LIN {X 0,Y 453.671,Z 73.472,A -85,B 0,C 180,E1 -8454.666,E2 -8454.666} C_VEL
LIN {X 0,Y 453.744,Z 73.459,A -85,B 0,C 180,E1 -8457.336,E2 -8457.336} C_VEL
LIN {X 0,Y 453.822,Z 73.438,A -85,B 0,C 180,E1 -8460,E2 -8460} C_VEL
LIN {X 0,Y 453.744,Z 73.457,A -85,B 0,C 180,E1 -8462.663,E2 -8462.663} C_VEL
LIN {X 0,Y 453.677,Z 73.469,A -85,B 0,C 180,E1 -8466.225,E2 -8466.225} C_VEL
LIN {X 0,Y 453.591,Z 73.469,A -85,B 0,C 180,E1 -8468.913,E2 -8468.913} C_VEL
LIN {X 0,Y 453.601,Z 73.475,A -85,B 0,C 180,E1 -8472.55,E2 -8472.55} C_VEL
LIN {X 0,Y 453.543,Z 73.483,A -85,B 0,C 180,E1 -8476.195,E2 -8476.195} C_VEL
LIN {X 0,Y 453.518,Z 73.478,A -85,B 0,C 180,E1 -8479.04,E2 -8479.04} C_VEL
LIN {X 0,Y 453.475,Z 73.495,A -85,B 0,C 180,E1 -8481.836,E2 -8481.836} C_VEL
LIN {X 0,Y 453.512,Z 73.492,A -85,B 0,C 180,E1 -8484.734,E2 -8484.734} C_VEL
LIN {X 0,Y 453.535,Z 73.478,A -85,B 0,C 180,E1 -8487.96,E2 -8487.96} C_VEL
LIN {X 0,Y 453.464,Z 73.497,A -85,B 0,C 180,E1 -8491.525,E2 -8491.525} C_VEL
LIN {X 0,Y 453.486,Z 73.489,A -85,B 0,C 180,E1 -8494.777,E2 -8494.777} C_VEL
LIN {X 0,Y 453.477,Z 73.498,A -85,B 0,C 180,E1 -8498.31,E2 -8498.31} C_VEL
LIN {X 0,Y 453.513,Z 73.488,A -85,B 0,C 180,E1 -8500.606,E2 -8500.606} C_VEL
LIN {X 0,Y 453.463,Z 73.501,A -85,B 0,C 180,E1 -8504.221,E2 -8504.221} C_VEL
LIN {X 0,Y 453.458,Z 73.476,A -85,B 0,C 180,E1 -8507.005,E2 -8507.005} C_VEL
LIN {X 0,Y 453.502,Z 73.493,A -85,B 0,C 180,E1 -8510.552,E2 -8510.552} C_VEL
LIN {X 0,Y 453.454,Z 73.495,A -85,B 0,C 180,E1 -8513.917,E2 -8513.917} C_VEL
LIN {X 0,Y 453.479,Z 73.493,A -85,B 0,C 180,E1 -8517.151,E2 -8517.151} C_VEL
LIN {X 0,Y 453.471,Z 73.488,A -85,B 0,C 180,E1 -8520.268,E2 -8520.268} C_VEL
LIN {X 0,Y 453.506,Z 73.494,A -85,B 0,C 180,E1 -8523.294,E2 -8523.294} C_VEL
LIN {X 0,Y 453.5,Z 73.496,A -85,B 0,C 180,E1 -8526.239,E2 -8526.239} C_VEL
LIN {X 0,Y 453.48,Z 73.498,A -85,B 0,C 180,E1 -8529.118,E2 -8529.118} C_VEL
LIN {X 0,Y 453.509,Z 73.497,A -85,B 0,C 180,E1 -8531.945,E2 -8531.945} C_VEL
LIN {X 0,Y 453.538,Z 73.491,A -85,B 0,C 180,E1 -8534.726,E2 -8534.726} C_VEL
LIN {X 0,Y 453.557,Z 73.488,A -85,B 0,C 180,E1 -8538.379,E2 -8538.379} C_VEL
LIN {X 0,Y 453.649,Z 73.478,A -85,B 0,C 180,E1 -8541.985,E2 -8541.985} C_VEL
LIN {X 0,Y 453.634,Z 73.479,A -85,B 0,C 180,E1 -8543.083,E2 -8543.083} C_VEL
LIN {X 0,Y 452.949,Z 73.565,A -85,B 0,C 180,E1 -8543.824,E2 -8543.824} C_VEL
LIN {X 0,Y 449.999,Z 73.934,A -85,B 0,C 180,E1 -8545.025,E2 -8545.025} C_VEL
LIN {X 0,Y 447.575,Z 74.234,A -85,B 0,C 180,E1 -8545.995,E2 -8545.995} C_VEL
LIN {X 0,Y 446.638,Z 74.352,A -85,B 0,C 180,E1 -8546.745,E2 -8546.745} C_VEL
LIN {X 0,Y 446.618,Z 74.353,A -85,B 0,C 180,E1 -8546.999,E2 -8546.999} C_VEL
LIN {X 0,Y 446.791,Z 74.332,A -85,B 0,C 180,E1 -8550,E2 -8550} C_VEL
LIN {X 0,Y 446.706,Z 74.344,A -85,B 0,C 180,E1 -8552.705,E2 -8552.705} C_VEL
LIN {X 0,Y 446.645,Z 74.351,A -85,B 0,C 180,E1 -8556.324,E2 -8556.324} C_VEL
LIN {X 0,Y 446.535,Z 74.365,A -85,B 0,C 180,E1 -8559.055,E2 -8559.055} C_VEL
LIN {X 0,Y 446.518,Z 74.367,A -85,B 0,C 180,E1 -8562.73,E2 -8562.73} C_VEL
LIN {X 0,Y 446.493,Z 74.371,A -85,B 0,C 180,E1 -8566.228,E2 -8566.228} C_VEL
LIN {X 0,Y 446.466,Z 74.371,A -85,B 0,C 180,E1 -8569.303,E2 -8569.303} C_VEL
LIN {X 0,Y 446.416,Z 74.381,A -85,B 0,C 180,E1 -8572.2,E2 -8572.2} C_VEL
LIN {X 0,Y 446.454,Z 74.371,A -85,B 0,C 180,E1 -8575.152,E2 -8575.152} C_VEL
LIN {X 0,Y 446.481,Z 74.364,A -85,B 0,C 180,E1 -8578.179,E2 -8578.179} C_VEL
LIN {X 0,Y 446.431,Z 74.378,A -85,B 0,C 180,E1 -8581.778,E2 -8581.778} C_VEL
LIN {X 0,Y 446.427,Z 74.353,A -85,B 0,C 180,E1 -8585.054,E2 -8585.054} C_VEL
LIN {X 0,Y 446.427,Z 74.377,A -85,B 0,C 180,E1 -8588.082,E2 -8588.082} C_VEL
LIN {X 0,Y 446.423,Z 74.361,A -85,B 0,C 180,E1 -8590.918,E2 -8590.918} C_VEL
LIN {X 0,Y 446.396,Z 74.367,A -85,B 0,C 180,E1 -8593.846,E2 -8593.846} C_VEL
LIN {X 0,Y 446.396,Z 74.377,A -85,B 0,C 180,E1 -8596.404,E2 -8596.404} C_VEL
LIN {X 0,Y 446.464,Z 74.367,A -85,B 0,C 180,E1 -8599.805,E2 -8599.805} C_VEL
LIN {X 0,Y 446.428,Z 74.374,A -85,B 0,C 180,E1 -8602.124,E2 -8602.124} C_VEL
LIN {X 0,Y 446.428,Z 74.367,A -85,B 0,C 180,E1 -8605.478,E2 -8605.478} C_VEL
LIN {X 0,Y 446.414,Z 74.377,A -85,B 0,C 180,E1 -8608.7,E2 -8608.7} C_VEL
LIN {X 0,Y 446.482,Z 74.357,A -85,B 0,C 180,E1 -8611.822,E2 -8611.822} C_VEL
LIN {X 0,Y 446.456,Z 74.369,A -85,B 0,C 180,E1 -8614.848,E2 -8614.848} C_VEL
LIN {X 0,Y 446.446,Z 74.371,A -85,B 0,C 180,E1 -8618.245,E2 -8618.245} C_VEL
LIN {X 0,Y 446.455,Z 74.356,A -85,B 0,C 180,E1 -8621.65,E2 -8621.65} C_VEL
LIN {X 0,Y 446.506,Z 74.366,A -85,B 0,C 180,E1 -8624.48,E2 -8624.48} C_VEL
LIN {X 0,Y 446.538,Z 74.357,A -85,B 0,C 180,E1 -8628.194,E2 -8628.194} C_VEL
LIN {X 0,Y 446.599,Z 74.341,A -85,B 0,C 180,E1 -8631.858,E2 -8631.858} C_VEL
LIN {X 0,Y 446.645,Z 74.349,A -85,B 0,C 180,E1 -8634.583,E2 -8634.583} C_VEL
LIN {X 0,Y 446.664,Z 74.335,A -85,B 0,C 180,E1 -8638.197,E2 -8638.197} C_VEL
LIN {X 0,Y 446.792,Z 74.312,A -85,B 0,C 180,E1 -8640,E2 -8640} C_VEL
LIN {X 0,Y 446.691,Z 74.337,A -85,B 0,C 180,E1 -8642.706,E2 -8642.706} C_VEL
LIN {X 0,Y 446.647,Z 74.344,A -85,B 0,C 180,E1 -8646.324,E2 -8646.324} C_VEL
LIN {X 0,Y 446.538,Z 74.346,A -85,B 0,C 180,E1 -8649.056,E2 -8649.056} C_VEL
LIN {X 0,Y 446.522,Z 74.357,A -85,B 0,C 180,E1 -8652.73,E2 -8652.73} C_VEL
LIN {X 0,Y 446.497,Z 74.359,A -85,B 0,C 180,E1 -8656.228,E2 -8656.228} C_VEL
LIN {X 0,Y 446.47,Z 74.354,A -85,B 0,C 180,E1 -8659.304,E2 -8659.304} C_VEL
LIN {X 0,Y 446.419,Z 74.372,A -85,B 0,C 180,E1 -8662.2,E2 -8662.2} C_VEL
LIN {X 0,Y 446.459,Z 74.367,A -85,B 0,C 180,E1 -8665.153,E2 -8665.153} C_VEL
LIN {X 0,Y 446.486,Z 74.358,A -85,B 0,C 180,E1 -8668.179,E2 -8668.179} C_VEL
LIN {X 0,Y 446.42,Z 74.373,A -85,B 0,C 180,E1 -8671.775,E2 -8671.775} C_VEL
LIN {X 0,Y 446.43,Z 74.364,A -85,B 0,C 180,E1 -8674.523,E2 -8674.523} C_VEL
LIN {X 0,Y 446.415,Z 74.375,A -85,B 0,C 180,E1 -8678.079,E2 -8678.079} C_VEL
LIN {X 0,Y 446.428,Z 74.373,A -85,B 0,C 180,E1 -8680.918,E2 -8680.918} C_VEL
LIN {X 0,Y 446.401,Z 74.376,A -85,B 0,C 180,E1 -8683.847,E2 -8683.847} C_VEL
LIN {X 0,Y 446.4,Z 74.381,A -85,B 0,C 180,E1 -8686.404,E2 -8686.404} C_VEL
LIN {X 0,Y 446.428,Z 74.361,A -85,B 0,C 180,E1 -8689.083,E2 -8689.083} C_VEL
LIN {X 0,Y 446.429,Z 74.376,A -85,B 0,C 180,E1 -8692.123,E2 -8692.123} C_VEL
LIN {X 0,Y 446.432,Z 74.37,A -85,B 0,C 180,E1 -8695.477,E2 -8695.477} C_VEL
LIN {X 0,Y 446.419,Z 74.377,A -85,B 0,C 180,E1 -8698.7,E2 -8698.7} C_VEL
LIN {X 0,Y 446.548,Z 74.569,A -85,B 0,C 180,E1 -8701.867,E2 -8701.867} C_VEL
LIN {X 0,Y 448.347,Z 84.511,A -85,B 0,C 180,E1 -8704.464,E2 -8704.464} C_VEL
LIN {X 0,Y 448.456,Z 88.047,A -85,B 0,C 180,E1 -8705.362,E2 -8705.362} C_VEL
LIN {X 0,Y 447.632,Z 102.965,A -85,B 0,C 180,E1 -8708.832,E2 -8708.832} C_VEL
LIN {X 0,Y 447.004,Z 115.084,A -85,B 0,C 180,E1 -8711.673,E2 -8711.673} C_VEL
LIN {X 0,Y 446.957,Z 117.073,A -85,B 0,C 180,E1 -8712.115,E2 -8712.115} C_VEL
LIN {X 0,Y 447.469,Z 120.446,A -85,B 0,C 180,E1 -8712.243,E2 -8712.243} C_VEL
LIN {X 0,Y 450.806,Z 140.583,A -85,B 0,C 180,E1 -8712.706,E2 -8712.706} C_VEL
LIN {X 0,Y 450.052,Z 221.953,A -85,B 0,C 180,E1 -8714.024,E2 -8714.024} C_VEL
LIN {X 0,Y 449.783,Z 231.85,A -85,B 0,C 180,E1 -8714.276,E2 -8714.276} C_VEL
LIN {X 0,Y 449.405,Z 241.826,A -85,B 0,C 180,E1 -8714.64,E2 -8714.64} C_VEL
LIN {X 0,Y 448.986,Z 252.191,A -85,B 0,C 180,E1 -8715.148,E2 -8715.148} C_VEL
LIN {X 0,Y 448.514,Z 261.326,A -85,B 0,C 180,E1 -8715.712,E2 -8715.712} C_VEL
LIN {X 0,Y 448.006,Z 270.323,A -85,B 0,C 180,E1 -8716.39,E2 -8716.39} C_VEL
LIN {X 0,Y 447.59,Z 278.193,A -85,B 0,C 180,E1 -8717.098,E2 -8717.098} C_VEL
LIN {X 0,Y 447.145,Z 286.451,A -85,B 0,C 180,E1 -8717.98,E2 -8717.98} C_VEL
LIN {X 0,Y 446.687,Z 293.671,A -85,B 0,C 180,E1 -8718.888,E2 -8718.888} C_VEL
LIN {X 0,Y 446.344,Z 299.873,A -85,B 0,C 180,E1 -8719.797,E2 -8719.797} C_VEL
LIN {X 0,Y 445.989,Z 306.41,A -85,B 0,C 180,E1 -8720.933,E2 -8720.933} C_VEL
LIN {X 0,Y 445.785,Z 310.912,A -85,B 0,C 180,E1 -8721.843,E2 -8721.843} C_VEL
LIN {X 0,Y 445.554,Z 316.557,A -85,B 0,C 180,E1 -8723.251,E2 -8723.251} C_VEL
LIN {X 0,Y 445.473,Z 320.725,A -85,B 0,C 180,E1 -8724.568,E2 -8724.568} C_VEL
LIN {X 0,Y 445.412,Z 323.089,A -85,B 0,C 180,E1 -8725.475,E2 -8725.475} C_VEL
LIN {X 0,Y 445.433,Z 326.273,A -85,B 0,C 180,E1 -8727.287,E2 -8727.287} C_VEL
LIN {X 0,Y 445.356,Z 327.327,A -85,B 0,C 180,E1 -8728.191,E2 -8728.191} C_VEL
LIN {X 0,Y 445.341,Z 327.914,A -85,B 0,C 180,E1 -8729.096,E2 -8729.096} C_VEL
LIN {X 0,Y 445.341,Z 327.914,A -85,B 0,C 180,E1 -8730.904,E2 -8730.904} C_VEL
LIN {X 0,Y 445.356,Z 327.327,A -85,B 0,C 180,E1 -8731.809,E2 -8731.809} C_VEL
LIN {X 0,Y 445.433,Z 326.273,A -85,B 0,C 180,E1 -8732.713,E2 -8732.713} C_VEL
LIN {X 0,Y 445.412,Z 323.089,A -85,B 0,C 180,E1 -8734.525,E2 -8734.525} C_VEL
LIN {X 0,Y 445.466,Z 318.987,A -85,B 0,C 180,E1 -8736.038,E2 -8736.038} C_VEL
LIN {X 0,Y 445.601,Z 314.742,A -85,B 0,C 180,E1 -8737.249,E2 -8737.249} C_VEL
LIN {X 0,Y 445.887,Z 308.722,A -85,B 0,C 180,E1 -8738.612,E2 -8738.612} C_VEL
LIN {X 0,Y 446.179,Z 302.625,A -85,B 0,C 180,E1 -8739.749,E2 -8739.749} C_VEL
LIN {X 0,Y 446.489,Z 296.924,A -85,B 0,C 180,E1 -8740.658,E2 -8740.658} C_VEL
LIN {X 0,Y 447.013,Z 288.37,A -85,B 0,C 180,E1 -8741.794,E2 -8741.794} C_VEL
LIN {X 0,Y 447.481,Z 280.189,A -85,B 0,C 180,E1 -8742.702,E2 -8742.702} C_VEL
LIN {X 0,Y 447.961,Z 271.759,A -85,B 0,C 180,E1 -8743.489,E2 -8743.489} C_VEL
LIN {X 0,Y 448.412,Z 262.957,A -85,B 0,C 180,E1 -8744.175,E2 -8744.175} C_VEL
LIN {X 0,Y 448.929,Z 253.198,A -85,B 0,C 180,E1 -8744.796,E2 -8744.796} C_VEL
LIN {X 0,Y 449.332,Z 244.402,A -85,B 0,C 180,E1 -8745.246,E2 -8745.246} C_VEL
LIN {X 0,Y 449.711,Z 234.473,A -85,B 0,C 180,E1 -8745.639,E2 -8745.639} C_VEL
LIN {X 0,Y 450.046,Z 224.618,A -85,B 0,C 180,E1 -8745.918,E2 -8745.918} C_VEL
LIN {X 0,Y 450.333,Z 200.656,A -85,B 0,C 180,E1 -8746.333,E2 -8746.333} C_VEL
LIN {X 0,Y 450.666,Z 138.88,A -85,B 0,C 180,E1 -8747.327,E2 -8747.327} C_VEL
LIN {X 0,Y 446.978,Z 117.536,A -85,B 0,C 180,E1 -8747.841,E2 -8747.841} C_VEL
LIN {X 0,Y 446.948,Z 116.116,A -85,B 0,C 180,E1 -8748.073,E2 -8748.073} C_VEL
LIN {X 0,Y 447.654,Z 103.185,A -85,B 0,C 180,E1 -8751.167,E2 -8751.167} C_VEL
LIN {X 0,Y 448.399,Z 89.526,A -85,B 0,C 180,E1 -8754.347,E2 -8754.347} C_VEL
LIN {X 0,Y 448.49,Z 85.556,A -85,B 0,C 180,E1 -8755.278,E2 -8755.278} C_VEL
LIN {X 0,Y 446.71,Z 75.373,A -85,B 0,C 180,E1 -8757.908,E2 -8757.908} C_VEL
LIN {X 0,Y 446.514,Z 74.374,A -85,B 0,C 180,E1 -8758.28,E2 -8758.28} C_VEL
LIN {X 0,Y 446.422,Z 74.373,A -85,B 0,C 180,E1 -8761.775,E2 -8761.775} C_VEL
LIN {X 0,Y 446.432,Z 74.371,A -85,B 0,C 180,E1 -8764.523,E2 -8764.523} C_VEL
LIN {X 0,Y 446.431,Z 74.373,A -85,B 0,C 180,E1 -8768.081,E2 -8768.081} C_VEL
LIN {X 0,Y 446.428,Z 74.362,A -85,B 0,C 180,E1 -8770.917,E2 -8770.917} C_VEL
LIN {X 0,Y 446.402,Z 74.378,A -85,B 0,C 180,E1 -8773.846,E2 -8773.846} C_VEL
LIN {X 0,Y 446.399,Z 74.376,A -85,B 0,C 180,E1 -8776.403,E2 -8776.403} C_VEL
LIN {X 0,Y 446.428,Z 74.374,A -85,B 0,C 180,E1 -8779.082,E2 -8779.082} C_VEL
LIN {X 0,Y 446.409,Z 74.375,A -85,B 0,C 180,E1 -8782.121,E2 -8782.121} C_VEL
LIN {X 0,Y 446.43,Z 74.364,A -85,B 0,C 180,E1 -8785.477,E2 -8785.477} C_VEL
LIN {X 0,Y 446.417,Z 74.377,A -85,B 0,C 180,E1 -8788.699,E2 -8788.699} C_VEL
LIN {X 0,Y 446.486,Z 74.358,A -85,B 0,C 180,E1 -8791.821,E2 -8791.821} C_VEL
LIN {X 0,Y 446.459,Z 74.367,A -85,B 0,C 180,E1 -8794.847,E2 -8794.847} C_VEL
LIN {X 0,Y 446.449,Z 74.371,A -85,B 0,C 180,E1 -8798.245,E2 -8798.245} C_VEL
LIN {X 0,Y 446.457,Z 74.352,A -85,B 0,C 180,E1 -8801.649,E2 -8801.649} C_VEL
LIN {X 0,Y 446.508,Z 74.365,A -85,B 0,C 180,E1 -8804.479,E2 -8804.479} C_VEL
LIN {X 0,Y 446.518,Z 74.358,A -85,B 0,C 180,E1 -8808.193,E2 -8808.193} C_VEL
LIN {X 0,Y 446.601,Z 74.34,A -85,B 0,C 180,E1 -8811.857,E2 -8811.857} C_VEL
LIN {X 0,Y 446.646,Z 74.348,A -85,B 0,C 180,E1 -8814.582,E2 -8814.582} C_VEL
LIN {X 0,Y 446.664,Z 74.335,A -85,B 0,C 180,E1 -8818.196,E2 -8818.196} C_VEL
LIN {X 0,Y 446.792,Z 74.312,A -85,B 0,C 180,E1 -8820,E2 -8820} C_VEL
LIN {X 0,Y 446.691,Z 74.336,A -85,B 0,C 180,E1 -8822.705,E2 -8822.705} C_VEL
LIN {X 0,Y 446.646,Z 74.344,A -85,B 0,C 180,E1 -8826.323,E2 -8826.323} C_VEL
LIN {X 0,Y 446.537,Z 74.348,A -85,B 0,C 180,E1 -8829.055,E2 -8829.055} C_VEL
LIN {X 0,Y 446.533,Z 74.356,A -85,B 0,C 180,E1 -8832.729,E2 -8832.729} C_VEL
LIN {X 0,Y 446.489,Z 74.362,A -85,B 0,C 180,E1 -8836.459,E2 -8836.459} C_VEL
LIN {X 0,Y 446.467,Z 74.356,A -85,B 0,C 180,E1 -8839.303,E2 -8839.303} C_VEL
LIN {X 0,Y 446.416,Z 74.373,A -85,B 0,C 180,E1 -8842.199,E2 -8842.199} C_VEL
LIN {X 0,Y 446.456,Z 74.369,A -85,B 0,C 180,E1 -8845.152,E2 -8845.152} C_VEL
LIN {X 0,Y 446.482,Z 74.357,A -85,B 0,C 180,E1 -8848.178,E2 -8848.178} C_VEL
LIN {X 0,Y 446.417,Z 74.374,A -85,B 0,C 180,E1 -8851.775,E2 -8851.775} C_VEL
LIN {X 0,Y 446.428,Z 74.367,A -85,B 0,C 180,E1 -8854.522,E2 -8854.522} C_VEL
LIN {X 0,Y 446.432,Z 74.374,A -85,B 0,C 180,E1 -8858.082,E2 -8858.082} C_VEL
LIN {X 0,Y 446.44,Z 74.369,A -85,B 0,C 180,E1 -8860.92,E2 -8860.92} C_VEL
LIN {X 0,Y 446.398,Z 74.378,A -85,B 0,C 180,E1 -8863.846,E2 -8863.846} C_VEL
LIN {X 0,Y 446.394,Z 74.363,A -85,B 0,C 180,E1 -8866.403,E2 -8866.403} C_VEL
LIN {X 0,Y 446.423,Z 74.361,A -85,B 0,C 180,E1 -8869.082,E2 -8869.082} C_VEL
LIN {X 0,Y 446.425,Z 74.38,A -85,B 0,C 180,E1 -8872.123,E2 -8872.123} C_VEL
LIN {X 0,Y 446.427,Z 74.357,A -85,B 0,C 180,E1 -8875.477,E2 -8875.477} C_VEL
LIN {X 0,Y 446.412,Z 74.376,A -85,B 0,C 180,E1 -8878.699,E2 -8878.699} C_VEL
LIN {X 0,Y 446.481,Z 74.364,A -85,B 0,C 180,E1 -8881.821,E2 -8881.821} C_VEL
LIN {X 0,Y 446.454,Z 74.371,A -85,B 0,C 180,E1 -8884.848,E2 -8884.848} C_VEL
LIN {X 0,Y 446.445,Z 74.375,A -85,B 0,C 180,E1 -8888.245,E2 -8888.245} C_VEL
LIN {X 0,Y 446.454,Z 74.376,A -85,B 0,C 180,E1 -8891.649,E2 -8891.649} C_VEL
LIN {X 0,Y 446.505,Z 74.367,A -85,B 0,C 180,E1 -8894.48,E2 -8894.48} C_VEL
LIN {X 0,Y 446.514,Z 74.366,A -85,B 0,C 180,E1 -8898.193,E2 -8898.193} C_VEL
LIN {X 0,Y 446.597,Z 74.357,A -85,B 0,C 180,E1 -8901.858,E2 -8901.858} C_VEL
LIN {X 0,Y 446.644,Z 74.351,A -85,B 0,C 180,E1 -8904.583,E2 -8904.583} C_VEL
LIN {X 0,Y 446.618,Z 74.353,A -85,B 0,C 180,E1 -8906.999,E2 -8906.999} C_VEL
LIN {X 0,Y 446.101,Z 74.421,A -85,B 0,C 180,E1 -8907.752,E2 -8907.752} C_VEL
LIN {X 0,Y 443.286,Z 74.776,A -85,B 0,C 180,E1 -8908.975,E2 -8908.975} C_VEL
LIN {X 0,Y 440.802,Z 75.085,A -85,B 0,C 180,E1 -8909.961,E2 -8909.961} C_VEL
LIN {X 0,Y 439.713,Z 75.217,A -85,B 0,C 180,E1 -8910.725,E2 -8910.725} C_VEL
LIN {X 0,Y 439.619,Z 75.226,A -85,B 0,C 180,E1 -8910.984,E2 -8910.984} C_VEL
LIN {X 0,Y 439.652,Z 75.222,A -85,B 0,C 180,E1 -8912.749,E2 -8912.749} C_VEL
LIN {X 0,Y 439.616,Z 75.228,A -85,B 0,C 180,E1 -8916.425,E2 -8916.425} C_VEL
LIN {X 0,Y 439.497,Z 75.242,A -85,B 0,C 180,E1 -8919.202,E2 -8919.202} C_VEL
LIN {X 0,Y 439.462,Z 75.246,A -85,B 0,C 180,E1 -8922.938,E2 -8922.938} C_VEL
LIN {X 0,Y 439.444,Z 75.249,A -85,B 0,C 180,E1 -8926.349,E2 -8926.349} C_VEL
LIN {X 0,Y 439.399,Z 75.252,A -85,B 0,C 180,E1 -8929.626,E2 -8929.626} C_VEL
LIN {X 0,Y 439.362,Z 75.258,A -85,B 0,C 180,E1 -8932.575,E2 -8932.575} C_VEL
LIN {X 0,Y 439.402,Z 75.251,A -85,B 0,C 180,E1 -8935.585,E2 -8935.585} C_VEL
LIN {X 0,Y 439.414,Z 75.239,A -85,B 0,C 180,E1 -8938.674,E2 -8938.674} C_VEL
LIN {X 0,Y 439.378,Z 75.256,A -85,B 0,C 180,E1 -8942.033,E2 -8942.033} C_VEL
LIN {X 0,Y 439.393,Z 75.231,A -85,B 0,C 180,E1 -8945.341,E2 -8945.341} C_VEL
LIN {X 0,Y 439.385,Z 75.251,A -85,B 0,C 180,E1 -8948.595,E2 -8948.595} C_VEL
LIN {X 0,Y 439.385,Z 75.23,A -85,B 0,C 180,E1 -8951.257,E2 -8951.257} C_VEL
LIN {X 0,Y 439.397,Z 75.243,A -85,B 0,C 180,E1 -8954.73,E2 -8954.73} C_VEL
LIN {X 0,Y 439.394,Z 75.248,A -85,B 0,C 180,E1 -8957.796,E2 -8957.796} C_VEL
LIN {X 0,Y 439.445,Z 75.239,A -85,B 0,C 180,E1 -8960.23,E2 -8960.23} C_VEL
LIN {X 0,Y 439.374,Z 75.25,A -85,B 0,C 180,E1 -8963.714,E2 -8963.714} C_VEL
LIN {X 0,Y 439.37,Z 75.25,A -85,B 0,C 180,E1 -8967.054,E2 -8967.054} C_VEL
LIN {X 0,Y 439.38,Z 75.25,A -85,B 0,C 180,E1 -8970.275,E2 -8970.275} C_VEL
LIN {X 0,Y 439.427,Z 75.239,A -85,B 0,C 180,E1 -8973.397,E2 -8973.397} C_VEL
LIN {X 0,Y 439.385,Z 75.252,A -85,B 0,C 180,E1 -8976.43,E2 -8976.43} C_VEL
LIN {X 0,Y 439.386,Z 75.241,A -85,B 0,C 180,E1 -8979.398,E2 -8979.398} C_VEL
LIN {X 0,Y 439.43,Z 75.234,A -85,B 0,C 180,E1 -8982.31,E2 -8982.31} C_VEL
LIN {X 0,Y 439.446,Z 75.243,A -85,B 0,C 180,E1 -8985.174,E2 -8985.174} C_VEL
LIN {X 0,Y 439.506,Z 75.234,A -85,B 0,C 180,E1 -8988.002,E2 -8988.002} C_VEL
LIN {X 0,Y 439.547,Z 75.218,A -85,B 0,C 180,E1 -8991.727,E2 -8991.727} C_VEL
LIN {X 0,Y 439.62,Z 75.225,A -85,B 0,C 180,E1 -8994.496,E2 -8994.496} C_VEL
LIN {X 0,Y 439.634,Z 75.21,A -85,B 0,C 180,E1 -8998.168,E2 -8998.168} C_VEL
LIN {X 0,Y 439.762,Z 75.187,A -85,B 0,C 180,E1 -9000,E2 -9000} C_VEL
LIN {X 0,Y 439.64,Z 75.215,A -85,B 0,C 180,E1 -9002.749,E2 -9002.749} C_VEL
LIN {X 0,Y 439.618,Z 75.218,A -85,B 0,C 180,E1 -9006.426,E2 -9006.426} C_VEL
LIN {X 0,Y 439.5,Z 75.222,A -85,B 0,C 180,E1 -9009.202,E2 -9009.202} C_VEL
LIN {X 0,Y 439.466,Z 75.236,A -85,B 0,C 180,E1 -9012.938,E2 -9012.938} C_VEL
LIN {X 0,Y 439.448,Z 75.236,A -85,B 0,C 180,E1 -9016.349,E2 -9016.349} C_VEL
LIN {X 0,Y 439.403,Z 75.237,A -85,B 0,C 180,E1 -9019.627,E2 -9019.627} C_VEL
LIN {X 0,Y 439.366,Z 75.251,A -85,B 0,C 180,E1 -9022.576,E2 -9022.576} C_VEL
LIN {X 0,Y 439.406,Z 75.239,A -85,B 0,C 180,E1 -9025.585,E2 -9025.585} C_VEL
LIN {X 0,Y 439.418,Z 75.24,A -85,B 0,C 180,E1 -9028.674,E2 -9028.674} C_VEL
LIN {X 0,Y 439.371,Z 75.25,A -85,B 0,C 180,E1 -9032.031,E2 -9032.031} C_VEL
LIN {X 0,Y 439.396,Z 75.248,A -85,B 0,C 180,E1 -9035.341,E2 -9035.341} C_VEL
LIN {X 0,Y 439.377,Z 75.255,A -85,B 0,C 180,E1 -9038.596,E2 -9038.596} C_VEL
LIN {X 0,Y 439.39,Z 75.25,A -85,B 0,C 180,E1 -9041.257,E2 -9041.257} C_VEL
LIN {X 0,Y 439.401,Z 75.248,A -85,B 0,C 180,E1 -9044.73,E2 -9044.73} C_VEL
LIN {X 0,Y 439.398,Z 75.249,A -85,B 0,C 180,E1 -9047.796,E2 -9047.796} C_VEL
LIN {X 0,Y 439.413,Z 75.235,A -85,B 0,C 180,E1 -9050.226,E2 -9050.226} C_VEL
LIN {X 0,Y 439.379,Z 75.252,A -85,B 0,C 180,E1 -9053.713,E2 -9053.713} C_VEL
LIN {X 0,Y 439.375,Z 75.252,A -85,B 0,C 180,E1 -9057.054,E2 -9057.054} C_VEL
LIN {X 0,Y 439.385,Z 75.25,A -85,B 0,C 180,E1 -9060.274,E2 -9060.274} C_VEL
LIN {X 0,Y 439.493,Z 75.468,A -85,B 0,C 180,E1 -9061.638,E2 -9061.638} C_VEL
LIN {X 0,Y 441.131,Z 84.371,A -85,B 0,C 180,E1 -9064.016,E2 -9064.016} C_VEL
LIN {X 0,Y 441.53,Z 88.646,A -85,B 0,C 180,E1 -9065.134,E2 -9065.134} C_VEL
LIN {X 0,Y 440.646,Z 103.836,A -85,B 0,C 180,E1 -9068.725,E2 -9068.725} C_VEL
LIN {X 0,Y 440.024,Z 114.898,A -85,B 0,C 180,E1 -9071.371,E2 -9071.371} C_VEL
LIN {X 0,Y 439.957,Z 116.884,A -85,B 0,C 180,E1 -9071.821,E2 -9071.821} C_VEL
LIN {X 0,Y 440.418,Z 119.708,A -85,B 0,C 180,E1 -9071.94,E2 -9071.94} C_VEL
LIN {X 0,Y 444.019,Z 140.746,A -85,B 0,C 180,E1 -9072.439,E2 -9072.439} C_VEL
LIN {X 0,Y 443.248,Z 221.763,A -85,B 0,C 180,E1 -9073.772,E2 -9073.772} C_VEL
LIN {X 0,Y 442.93,Z 232.534,A -85,B 0,C 180,E1 -9074.056,E2 -9074.056} C_VEL
LIN {X 0,Y 442.574,Z 241.636,A -85,B 0,C 180,E1 -9074.397,E2 -9074.397} C_VEL
LIN {X 0,Y 442.132,Z 252,A -85,B 0,C 180,E1 -9074.913,E2 -9074.913} C_VEL
LIN {X 0,Y 441.632,Z 261.135,A -85,B 0,C 180,E1 -9075.485,E2 -9075.485} C_VEL
LIN {X 0,Y 441.1,Z 270.133,A -85,B 0,C 180,E1 -9076.173,E2 -9076.173} C_VEL
LIN {X 0,Y 440.602,Z 278.383,A -85,B 0,C 180,E1 -9076.93,E2 -9076.93} C_VEL
LIN {X 0,Y 440.188,Z 286.26,A -85,B 0,C 180,E1 -9077.787,E2 -9077.787} C_VEL
LIN {X 0,Y 439.705,Z 293.48,A -85,B 0,C 180,E1 -9078.709,E2 -9078.709} C_VEL
LIN {X 0,Y 439.332,Z 299.682,A -85,B 0,C 180,E1 -9079.632,E2 -9079.632} C_VEL
LIN {X 0,Y 438.961,Z 306.219,A -85,B 0,C 180,E1 -9080.787,E2 -9080.787} C_VEL
LIN {X 0,Y 438.738,Z 310.721,A -85,B 0,C 180,E1 -9081.711,E2 -9081.711} C_VEL
LIN {X 0,Y 438.493,Z 316.211,A -85,B 0,C 180,E1 -9083.096,E2 -9083.096} C_VEL
LIN {X 0,Y 438.371,Z 320.534,A -85,B 0,C 180,E1 -9084.48,E2 -9084.48} C_VEL
LIN {X 0,Y 438.341,Z 322.899,A -85,B 0,C 180,E1 -9085.402,E2 -9085.402} C_VEL
LIN {X 0,Y 438.341,Z 326.082,A -85,B 0,C 180,E1 -9087.243,E2 -9087.243} C_VEL
LIN {X 0,Y 438.279,Z 327.137,A -85,B 0,C 180,E1 -9088.162,E2 -9088.162} C_VEL
LIN {X 0,Y 438.254,Z 327.724,A -85,B 0,C 180,E1 -9089.081,E2 -9089.081} C_VEL
LIN {X 0,Y 438.254,Z 327.724,A -85,B 0,C 180,E1 -9090.919,E2 -9090.919} C_VEL
LIN {X 0,Y 438.279,Z 327.137,A -85,B 0,C 180,E1 -9091.838,E2 -9091.838} C_VEL
LIN {X 0,Y 438.341,Z 326.082,A -85,B 0,C 180,E1 -9092.757,E2 -9092.757} C_VEL
LIN {X 0,Y 438.341,Z 322.899,A -85,B 0,C 180,E1 -9094.598,E2 -9094.598} C_VEL
LIN {X 0,Y 438.422,Z 318.101,A -85,B 0,C 180,E1 -9096.342,E2 -9096.342} C_VEL
LIN {X 0,Y 438.633,Z 312.636,A -85,B 0,C 180,E1 -9097.827,E2 -9097.827} C_VEL
LIN {X 0,Y 438.885,Z 307.375,A -85,B 0,C 180,E1 -9098.982,E2 -9098.982} C_VEL
LIN {X 0,Y 439.216,Z 301.057,A -85,B 0,C 180,E1 -9100.138,E2 -9100.138} C_VEL
LIN {X 0,Y 439.572,Z 295.106,A -85,B 0,C 180,E1 -9101.061,E2 -9101.061} C_VEL
LIN {X 0,Y 440.052,Z 288.179,A -85,B 0,C 180,E1 -9101.983,E2 -9101.983} C_VEL
LIN {X 0,Y 440.538,Z 279.998,A -85,B 0,C 180,E1 -9102.906,E2 -9102.906} C_VEL
LIN {X 0,Y 441.015,Z 272.013,A -85,B 0,C 180,E1 -9103.666,E2 -9103.666} C_VEL
LIN {X 0,Y 441.505,Z 262.766,A -85,B 0,C 180,E1 -9104.402,E2 -9104.402} C_VEL
LIN {X 0,Y 442.048,Z 253.007,A -85,B 0,C 180,E1 -9105.031,E2 -9105.031} C_VEL
LIN {X 0,Y 442.495,Z 244.212,A -85,B 0,C 180,E1 -9105.487,E2 -9105.487} C_VEL
LIN {X 0,Y 442.878,Z 234.283,A -85,B 0,C 180,E1 -9105.887,E2 -9105.887} C_VEL
LIN {X 0,Y 443.22,Z 224.427,A -85,B 0,C 180,E1 -9106.17,E2 -9106.17} C_VEL
LIN {X 0,Y 443.552,Z 199.431,A -85,B 0,C 180,E1 -9106.607,E2 -9106.607} C_VEL
LIN {X 0,Y 443.878,Z 139.616,A -85,B 0,C 180,E1 -9107.586,E2 -9107.586} C_VEL
LIN {X 0,Y 439.962,Z 117.129,A -85,B 0,C 180,E1 -9108.15,E2 -9108.15} C_VEL
LIN {X 0,Y 439.975,Z 115.943,A -85,B 0,C 180,E1 -9108.366,E2 -9108.366} C_VEL
LIN {X 0,Y 440.664,Z 104.047,A -85,B 0,C 180,E1 -9111.274,E2 -9111.274} C_VEL
LIN {X 0,Y 441.44,Z 90.665,A -85,B 0,C 180,E1 -9114.452,E2 -9114.452} C_VEL
LIN {X 0,Y 441.487,Z 86.469,A -85,B 0,C 180,E1 -9115.455,E2 -9115.455} C_VEL
LIN {X 0,Y 439.782,Z 76.789,A -85,B 0,C 180,E1 -9117.996,E2 -9117.996} C_VEL
LIN {X 0,Y 439.443,Z 75.267,A -85,B 0,C 180,E1 -9118.473,E2 -9118.473} C_VEL
LIN {X 0,Y 439.372,Z 75.25,A -85,B 0,C 180,E1 -9122.03,E2 -9122.03} C_VEL
LIN {X 0,Y 439.398,Z 75.243,A -85,B 0,C 180,E1 -9125.34,E2 -9125.34} C_VEL
LIN {X 0,Y 439.384,Z 75.248,A -85,B 0,C 180,E1 -9128.595,E2 -9128.595} C_VEL
LIN {X 0,Y 439.39,Z 75.241,A -85,B 0,C 180,E1 -9131.256,E2 -9131.256} C_VEL
LIN {X 0,Y 439.401,Z 75.247,A -85,B 0,C 180,E1 -9134.729,E2 -9134.729} C_VEL
LIN {X 0,Y 439.397,Z 75.251,A -85,B 0,C 180,E1 -9137.795,E2 -9137.795} C_VEL
LIN {X 0,Y 439.396,Z 75.242,A -85,B 0,C 180,E1 -9140.224,E2 -9140.224} C_VEL
LIN {X 0,Y 439.375,Z 75.25,A -85,B 0,C 180,E1 -9143.712,E2 -9143.712} C_VEL
LIN {X 0,Y 439.374,Z 75.249,A -85,B 0,C 180,E1 -9147.054,E2 -9147.054} C_VEL
LIN {X 0,Y 439.383,Z 75.251,A -85,B 0,C 180,E1 -9150.274,E2 -9150.274} C_VEL
LIN {X 0,Y 439.429,Z 75.235,A -85,B 0,C 180,E1 -9153.396,E2 -9153.396} C_VEL
LIN {X 0,Y 439.388,Z 75.251,A -85,B 0,C 180,E1 -9156.429,E2 -9156.429} C_VEL
LIN {X 0,Y 439.389,Z 75.241,A -85,B 0,C 180,E1 -9159.397,E2 -9159.397} C_VEL
LIN {X 0,Y 439.431,Z 75.231,A -85,B 0,C 180,E1 -9162.309,E2 -9162.309} C_VEL
LIN {X 0,Y 439.448,Z 75.241,A -85,B 0,C 180,E1 -9165.174,E2 -9165.174} C_VEL
LIN {X 0,Y 439.484,Z 75.237,A -85,B 0,C 180,E1 -9168.001,E2 -9168.001} C_VEL
LIN {X 0,Y 439.548,Z 75.217,A -85,B 0,C 180,E1 -9171.726,E2 -9171.726} C_VEL
LIN {X 0,Y 439.621,Z 75.224,A -85,B 0,C 180,E1 -9174.495,E2 -9174.495} C_VEL
LIN {X 0,Y 439.634,Z 75.211,A -85,B 0,C 180,E1 -9178.167,E2 -9178.167} C_VEL
LIN {X 0,Y 439.762,Z 75.187,A -85,B 0,C 180,E1 -9180,E2 -9180} C_VEL
LIN {X 0,Y 439.64,Z 75.214,A -85,B 0,C 180,E1 -9182.748,E2 -9182.748} C_VEL
LIN {X 0,Y 439.617,Z 75.219,A -85,B 0,C 180,E1 -9186.425,E2 -9186.425} C_VEL
LIN {X 0,Y 439.5,Z 75.224,A -85,B 0,C 180,E1 -9189.201,E2 -9189.201} C_VEL
LIN {X 0,Y 439.503,Z 75.232,A -85,B 0,C 180,E1 -9192.726,E2 -9192.726} C_VEL
LIN {X 0,Y 439.446,Z 75.239,A -85,B 0,C 180,E1 -9196.348,E2 -9196.348} C_VEL
LIN {X 0,Y 439.401,Z 75.238,A -85,B 0,C 180,E1 -9199.626,E2 -9199.626} C_VEL
LIN {X 0,Y 439.363,Z 75.253,A -85,B 0,C 180,E1 -9202.575,E2 -9202.575} C_VEL
LIN {X 0,Y 439.403,Z 75.242,A -85,B 0,C 180,E1 -9205.584,E2 -9205.584} C_VEL
LIN {X 0,Y 439.415,Z 75.24,A -85,B 0,C 180,E1 -9208.673,E2 -9208.673} C_VEL
LIN {X 0,Y 439.368,Z 75.252,A -85,B 0,C 180,E1 -9212.03,E2 -9212.03} C_VEL
LIN {X 0,Y 439.394,Z 75.247,A -85,B 0,C 180,E1 -9215.34,E2 -9215.34} C_VEL
LIN {X 0,Y 439.392,Z 75.255,A -85,B 0,C 180,E1 -9218.593,E2 -9218.593} C_VEL
LIN {X 0,Y 439.395,Z 75.246,A -85,B 0,C 180,E1 -9221.258,E2 -9221.258} C_VEL
LIN {X 0,Y 439.398,Z 75.247,A -85,B 0,C 180,E1 -9224.729,E2 -9224.729} C_VEL
LIN {X 0,Y 439.392,Z 75.224,A -85,B 0,C 180,E1 -9227.795,E2 -9227.795} C_VEL
LIN {X 0,Y 439.426,Z 75.24,A -85,B 0,C 180,E1 -9230.228,E2 -9230.228} C_VEL
LIN {X 0,Y 439.374,Z 75.252,A -85,B 0,C 180,E1 -9233.713,E2 -9233.713} C_VEL
LIN {X 0,Y 439.369,Z 75.25,A -85,B 0,C 180,E1 -9237.054,E2 -9237.054} C_VEL
LIN {X 0,Y 439.378,Z 75.242,A -85,B 0,C 180,E1 -9240.274,E2 -9240.274} C_VEL
LIN {X 0,Y 439.426,Z 75.249,A -85,B 0,C 180,E1 -9243.396,E2 -9243.396} C_VEL
LIN {X 0,Y 439.384,Z 75.254,A -85,B 0,C 180,E1 -9246.43,E2 -9246.43} C_VEL
LIN {X 0,Y 439.386,Z 75.256,A -85,B 0,C 180,E1 -9249.397,E2 -9249.397} C_VEL
LIN {X 0,Y 439.428,Z 75.248,A -85,B 0,C 180,E1 -9252.309,E2 -9252.309} C_VEL
LIN {X 0,Y 439.446,Z 75.248,A -85,B 0,C 180,E1 -9255.174,E2 -9255.174} C_VEL
LIN {X 0,Y 439.48,Z 75.243,A -85,B 0,C 180,E1 -9258.001,E2 -9258.001} C_VEL
LIN {X 0,Y 439.545,Z 75.236,A -85,B 0,C 180,E1 -9261.726,E2 -9261.726} C_VEL
LIN {X 0,Y 439.619,Z 75.226,A -85,B 0,C 180,E1 -9264.496,E2 -9264.496} C_VEL
LIN {X 0,Y 439.633,Z 75.223,A -85,B 0,C 180,E1 -9268.168,E2 -9268.168} C_VEL
LIN {X 0,Y 439.761,Z 75.208,A -85,B 0,C 180,E1 -9270,E2 -9270} C_VEL
LIN {X 0,Y 439.619,Z 75.226,A -85,B 0,C 180,E1 -9270.984,E2 -9270.984} C_VEL
LIN {X 0,Y 438.902,Z 75.314,A -85,B 0,C 180,E1 -9271.748,E2 -9271.748} C_VEL
LIN {X 0,Y 435.923,Z 75.687,A -85,B 0,C 180,E1 -9272.987,E2 -9272.987} C_VEL
LIN {X 0,Y 433.471,Z 75.993,A -85,B 0,C 180,E1 -9273.987,E2 -9273.987} C_VEL
LIN {X 0,Y 432.498,Z 76.115,A -85,B 0,C 180,E1 -9274.762,E2 -9274.762} C_VEL
LIN {X 0,Y 432.461,Z 76.116,A -85,B 0,C 180,E1 -9275.024,E2 -9275.024} C_VEL
LIN {X 0,Y 432.582,Z 76.102,A -85,B 0,C 180,E1 -9277.679,E2 -9277.679} C_VEL
LIN {X 0,Y 432.39,Z 76.126,A -85,B 0,C 180,E1 -9281.247,E2 -9281.247} C_VEL
LIN {X 0,Y 432.372,Z 76.129,A -85,B 0,C 180,E1 -9284.112,E2 -9284.112} C_VEL
LIN {X 0,Y 432.394,Z 76.125,A -85,B 0,C 180,E1 -9287.012,E2 -9287.012} C_VEL
LIN {X 0,Y 432.336,Z 76.134,A -85,B 0,C 180,E1 -9289.96,E2 -9289.96} C_VEL
LIN {X 0,Y 432.316,Z 76.134,A -85,B 0,C 180,E1 -9292.964,E2 -9292.964} C_VEL
LIN {X 0,Y 432.361,Z 76.131,A -85,B 0,C 180,E1 -9296.033,E2 -9296.033} C_VEL
LIN {X 0,Y 432.339,Z 76.117,A -85,B 0,C 180,E1 -9299.188,E2 -9299.188} C_VEL
LIN {X 0,Y 432.324,Z 76.13,A -85,B 0,C 180,E1 -9302.443,E2 -9302.443} C_VEL
LIN {X 0,Y 432.342,Z 76.113,A -85,B 0,C 180,E1 -9305.632,E2 -9305.632} C_VEL
LIN {X 0,Y 432.347,Z 76.127,A -85,B 0,C 180,E1 -9308.716,E2 -9308.716} C_VEL
LIN {X 0,Y 432.329,Z 76.103,A -85,B 0,C 180,E1 -9311.797,E2 -9311.797} C_VEL
LIN {X 0,Y 432.33,Z 76.123,A -85,B 0,C 180,E1 -9314.348,E2 -9314.348} C_VEL
LIN {X 0,Y 432.317,Z 76.133,A -85,B 0,C 180,E1 -9317.016,E2 -9317.016} C_VEL
LIN {X 0,Y 432.352,Z 76.124,A -85,B 0,C 180,E1 -9319.818,E2 -9319.818} C_VEL
LIN {X 0,Y 432.314,Z 76.137,A -85,B 0,C 180,E1 -9323.023,E2 -9323.023} C_VEL
LIN {X 0,Y 432.357,Z 76.117,A -85,B 0,C 180,E1 -9325.997,E2 -9325.997} C_VEL
LIN {X 0,Y 432.345,Z 76.129,A -85,B 0,C 180,E1 -9329.49,E2 -9329.49} C_VEL
LIN {X 0,Y 432.39,Z 76.111,A -85,B 0,C 180,E1 -9332.929,E2 -9332.929} C_VEL
LIN {X 0,Y 432.37,Z 76.124,A -85,B 0,C 180,E1 -9336.024,E2 -9336.024} C_VEL
LIN {X 0,Y 432.348,Z 76.12,A -85,B 0,C 180,E1 -9339.047,E2 -9339.047} C_VEL
LIN {X 0,Y 432.376,Z 76.11,A -85,B 0,C 180,E1 -9342.012,E2 -9342.012} C_VEL
LIN {X 0,Y 432.394,Z 76.124,A -85,B 0,C 180,E1 -9344.927,E2 -9344.927} C_VEL
LIN {X 0,Y 432.48,Z 76.107,A -85,B 0,C 180,E1 -9347.805,E2 -9347.805} C_VEL
LIN {X 0,Y 432.491,Z 76.096,A -85,B 0,C 180,E1 -9351.591,E2 -9351.591} C_VEL
LIN {X 0,Y 432.597,Z 76.101,A -85,B 0,C 180,E1 -9354.407,E2 -9354.407} C_VEL
LIN {X 0,Y 432.603,Z 76.086,A -85,B 0,C 180,E1 -9358.139,E2 -9358.139} C_VEL
LIN {X 0,Y 432.732,Z 76.062,A -85,B 0,C 180,E1 -9360.001,E2 -9360.001} C_VEL
LIN {X 0,Y 432.592,Z 76.093,A -85,B 0,C 180,E1 -9362.794,E2 -9362.794} C_VEL
LIN {X 0,Y 432.573,Z 76.095,A -85,B 0,C 180,E1 -9366.531,E2 -9366.531} C_VEL
LIN {X 0,Y 432.443,Z 76.099,A -85,B 0,C 180,E1 -9369.354,E2 -9369.354} C_VEL
LIN {X 0,Y 432.431,Z 76.112,A -85,B 0,C 180,E1 -9372.804,E2 -9372.804} C_VEL
LIN {X 0,Y 432.413,Z 76.112,A -85,B 0,C 180,E1 -9376.479,E2 -9376.479} C_VEL
LIN {X 0,Y 432.34,Z 76.12,A -85,B 0,C 180,E1 -9379.961,E2 -9379.961} C_VEL
LIN {X 0,Y 432.32,Z 76.132,A -85,B 0,C 180,E1 -9382.965,E2 -9382.965} C_VEL
LIN {X 0,Y 432.365,Z 76.113,A -85,B 0,C 180,E1 -9386.033,E2 -9386.033} C_VEL
LIN {X 0,Y 432.344,Z 76.128,A -85,B 0,C 180,E1 -9389.188,E2 -9389.188} C_VEL
LIN {X 0,Y 432.324,Z 76.13,A -85,B 0,C 180,E1 -9392.443,E2 -9392.443} C_VEL
LIN {X 0,Y 432.346,Z 76.124,A -85,B 0,C 180,E1 -9395.632,E2 -9395.632} C_VEL
LIN {X 0,Y 432.339,Z 76.13,A -85,B 0,C 180,E1 -9398.714,E2 -9398.714} C_VEL
LIN {X 0,Y 432.335,Z 76.128,A -85,B 0,C 180,E1 -9401.798,E2 -9401.798} C_VEL
LIN {X 0,Y 432.335,Z 76.129,A -85,B 0,C 180,E1 -9404.348,E2 -9404.348} C_VEL
LIN {X 0,Y 432.322,Z 76.132,A -85,B 0,C 180,E1 -9407.016,E2 -9407.016} C_VEL
LIN {X 0,Y 432.335,Z 76.114,A -85,B 0,C 180,E1 -9409.821,E2 -9409.821} C_VEL
LIN {X 0,Y 432.317,Z 76.131,A -85,B 0,C 180,E1 -9413.023,E2 -9413.023} C_VEL
LIN {X 0,Y 432.362,Z 76.127,A -85,B 0,C 180,E1 -9415.997,E2 -9415.997} C_VEL
LIN {X 0,Y 432.35,Z 76.133,A -85,B 0,C 180,E1 -9419.49,E2 -9419.49} C_VEL
LIN {X 0,Y 432.429,Z 76.256,A -85,B 0,C 180,E1 -9421.358,E2 -9421.358} C_VEL
LIN {X 0,Y 434.238,Z 86.185,A -85,B 0,C 180,E1 -9424.088,E2 -9424.088} C_VEL
LIN {X 0,Y 434.546,Z 90.21,A -85,B 0,C 180,E1 -9425.134,E2 -9425.134} C_VEL
LIN {X 0,Y 433.665,Z 104.707,A -85,B 0,C 180,E1 -9428.615,E2 -9428.615} C_VEL
LIN {X 0,Y 432.973,Z 116.695,A -85,B 0,C 180,E1 -9431.517,E2 -9431.517} C_VEL
LIN {X 0,Y 433.398,Z 119.37,A -85,B 0,C 180,E1 -9431.634,E2 -9431.634} C_VEL
LIN {X 0,Y 437.239,Z 141.453,A -85,B 0,C 180,E1 -9432.173,E2 -9432.173} C_VEL
LIN {X 0,Y 436.448,Z 221.573,A -85,B 0,C 180,E1 -9433.512,E2 -9433.512} C_VEL
LIN {X 0,Y 436.138,Z 231.469,A -85,B 0,C 180,E1 -9433.771,E2 -9433.771} C_VEL
LIN {X 0,Y 435.729,Z 241.445,A -85,B 0,C 180,E1 -9434.146,E2 -9434.146} C_VEL
LIN {X 0,Y 435.304,Z 250.802,A -85,B 0,C 180,E1 -9434.61,E2 -9434.61} C_VEL
LIN {X 0,Y 434.737,Z 260.944,A -85,B 0,C 180,E1 -9435.249,E2 -9435.249} C_VEL
LIN {X 0,Y 434.191,Z 269.942,A -85,B 0,C 180,E1 -9435.948,E2 -9435.948} C_VEL
LIN {X 0,Y 433.631,Z 278.62,A -85,B 0,C 180,E1 -9436.761,E2 -9436.761} C_VEL
LIN {X 0,Y 433.234,Z 286.069,A -85,B 0,C 180,E1 -9437.588,E2 -9437.588} C_VEL
LIN {X 0,Y 432.731,Z 293.289,A -85,B 0,C 180,E1 -9438.524,E2 -9438.524} C_VEL
LIN {X 0,Y 432.291,Z 299.49,A -85,B 0,C 180,E1 -9439.461,E2 -9439.461} C_VEL
LIN {X 0,Y 431.907,Z 306.028,A -85,B 0,C 180,E1 -9440.635,E2 -9440.635} C_VEL
LIN {X 0,Y 431.68,Z 310.53,A -85,B 0,C 180,E1 -9441.574,E2 -9441.574} C_VEL
LIN {X 0,Y 431.413,Z 316.02,A -85,B 0,C 180,E1 -9442.982,E2 -9442.982} C_VEL
LIN {X 0,Y 431.274,Z 320.342,A -85,B 0,C 180,E1 -9444.389,E2 -9444.389} C_VEL
LIN {X 0,Y 431.27,Z 322.709,A -85,B 0,C 180,E1 -9445.326,E2 -9445.326} C_VEL
LIN {X 0,Y 431.236,Z 325.891,A -85,B 0,C 180,E1 -9447.198,E2 -9447.198} C_VEL
LIN {X 0,Y 431.203,Z 326.947,A -85,B 0,C 180,E1 -9448.132,E2 -9448.132} C_VEL
LIN {X 0,Y 431.171,Z 327.534,A -85,B 0,C 180,E1 -9449.066,E2 -9449.066} C_VEL
LIN {X 0,Y 431.171,Z 327.534,A -85,B 0,C 180,E1 -9450.934,E2 -9450.934} C_VEL
LIN {X 0,Y 431.203,Z 326.947,A -85,B 0,C 180,E1 -9451.868,E2 -9451.868} C_VEL
LIN {X 0,Y 431.187,Z 324.504,A -85,B 0,C 180,E1 -9453.738,E2 -9453.738} C_VEL
LIN {X 0,Y 431.291,Z 321.56,A -85,B 0,C 180,E1 -9455.142,E2 -9455.142} C_VEL
LIN {X 0,Y 431.377,Z 317.573,A -85,B 0,C 180,E1 -9456.548,E2 -9456.548} C_VEL
LIN {X 0,Y 431.565,Z 312.445,A -85,B 0,C 180,E1 -9457.957,E2 -9457.957} C_VEL
LIN {X 0,Y 431.833,Z 307.183,A -85,B 0,C 180,E1 -9459.13,E2 -9459.13} C_VEL
LIN {X 0,Y 432.193,Z 300.866,A -85,B 0,C 180,E1 -9460.304,E2 -9460.304} C_VEL
LIN {X 0,Y 432.586,Z 294.915,A -85,B 0,C 180,E1 -9461.242,E2 -9461.242} C_VEL
LIN {X 0,Y 433.08,Z 287.988,A -85,B 0,C 180,E1 -9462.179,E2 -9462.179} C_VEL
LIN {X 0,Y 433.584,Z 279.807,A -85,B 0,C 180,E1 -9463.116,E2 -9463.116} C_VEL
LIN {X 0,Y 434.117,Z 271.119,A -85,B 0,C 180,E1 -9463.95,E2 -9463.95} C_VEL
LIN {X 0,Y 434.613,Z 262.575,A -85,B 0,C 180,E1 -9464.635,E2 -9464.635} C_VEL
LIN {X 0,Y 435.173,Z 252.816,A -85,B 0,C 180,E1 -9465.275,E2 -9465.275} C_VEL
LIN {X 0,Y 435.696,Z 242.733,A -85,B 0,C 180,E1 -9465.795,E2 -9465.795} C_VEL
LIN {X 0,Y 436.086,Z 233.218,A -85,B 0,C 180,E1 -9466.171,E2 -9466.171} C_VEL
LIN {X 0,Y 436.415,Z 222.904,A -85,B 0,C 180,E1 -9466.459,E2 -9466.459} C_VEL
LIN {X 0,Y 437.165,Z 153.709,A -85,B 0,C 180,E1 -9467.624,E2 -9467.624} C_VEL
LIN {X 0,Y 437.058,Z 140.003,A -85,B 0,C 180,E1 -9467.859,E2 -9467.859} C_VEL
LIN {X 0,Y 433.003,Z 117.024,A -85,B 0,C 180,E1 -9468.447,E2 -9468.447} C_VEL
LIN {X 0,Y 432.989,Z 115.756,A -85,B 0,C 180,E1 -9468.673,E2 -9468.673} C_VEL
LIN {X 0,Y 433.718,Z 103.88,A -85,B 0,C 180,E1 -9471.632,E2 -9471.632} C_VEL
LIN {X 0,Y 434.557,Z 90.531,A -85,B 0,C 180,E1 -9474.866,E2 -9474.866} C_VEL
LIN {X 0,Y 434.284,Z 86.328,A -85,B 0,C 180,E1 -9475.909,E2 -9475.909} C_VEL
LIN {X 0,Y 432.81,Z 78.161,A -85,B 0,C 180,E1 -9478.093,E2 -9478.093} C_VEL
LIN {X 0,Y 432.392,Z 76.145,A -85,B 0,C 180,E1 -9478.704,E2 -9478.704} C_VEL
LIN {X 0,Y 432.324,Z 76.132,A -85,B 0,C 180,E1 -9481.346,E2 -9481.346} C_VEL
LIN {X 0,Y 432.343,Z 76.125,A -85,B 0,C 180,E1 -9484.677,E2 -9484.677} C_VEL
LIN {X 0,Y 432.346,Z 76.127,A -85,B 0,C 180,E1 -9488.149,E2 -9488.149} C_VEL
LIN {X 0,Y 432.335,Z 76.124,A -85,B 0,C 180,E1 -9491.602,E2 -9491.602} C_VEL
LIN {X 0,Y 432.335,Z 76.127,A -85,B 0,C 180,E1 -9494.347,E2 -9494.347} C_VEL
LIN {X 0,Y 432.321,Z 76.133,A -85,B 0,C 180,E1 -9497.015,E2 -9497.015} C_VEL
LIN {X 0,Y 432.334,Z 76.123,A -85,B 0,C 180,E1 -9499.82,E2 -9499.82} C_VEL
LIN {X 0,Y 432.308,Z 76.137,A -85,B 0,C 180,E1 -9503.022,E2 -9503.022} C_VEL
LIN {X 0,Y 432.361,Z 76.114,A -85,B 0,C 180,E1 -9505.996,E2 -9505.996} C_VEL
LIN {X 0,Y 432.349,Z 76.128,A -85,B 0,C 180,E1 -9509.489,E2 -9509.489} C_VEL
LIN {X 0,Y 432.392,Z 76.11,A -85,B 0,C 180,E1 -9512.928,E2 -9512.928} C_VEL
LIN {X 0,Y 432.373,Z 76.122,A -85,B 0,C 180,E1 -9516.023,E2 -9516.023} C_VEL
LIN {X 0,Y 432.351,Z 76.12,A -85,B 0,C 180,E1 -9519.046,E2 -9519.046} C_VEL
LIN {X 0,Y 432.378,Z 76.106,A -85,B 0,C 180,E1 -9522.011,E2 -9522.011} C_VEL
LIN {X 0,Y 432.396,Z 76.121,A -85,B 0,C 180,E1 -9524.926,E2 -9524.926} C_VEL
LIN {X 0,Y 432.46,Z 76.11,A -85,B 0,C 180,E1 -9527.803,E2 -9527.803} C_VEL
LIN {X 0,Y 432.492,Z 76.095,A -85,B 0,C 180,E1 -9531.59,E2 -9531.59} C_VEL
LIN {X 0,Y 432.598,Z 76.1,A -85,B 0,C 180,E1 -9534.406,E2 -9534.406} C_VEL
LIN {X 0,Y 432.603,Z 76.087,A -85,B 0,C 180,E1 -9538.138,E2 -9538.138} C_VEL
LIN {X 0,Y 432.732,Z 76.062,A -85,B 0,C 180,E1 -9539.999,E2 -9539.999} C_VEL
LIN {X 0,Y 432.592,Z 76.092,A -85,B 0,C 180,E1 -9542.793,E2 -9542.793} C_VEL
LIN {X 0,Y 432.572,Z 76.096,A -85,B 0,C 180,E1 -9546.53,E2 -9546.53} C_VEL
LIN {X 0,Y 432.443,Z 76.1,A -85,B 0,C 180,E1 -9549.353,E2 -9549.353} C_VEL
LIN {X 0,Y 432.444,Z 76.111,A -85,B 0,C 180,E1 -9552.811,E2 -9552.811} C_VEL
LIN {X 0,Y 432.411,Z 76.115,A -85,B 0,C 180,E1 -9556.478,E2 -9556.478} C_VEL
LIN {X 0,Y 432.337,Z 76.119,A -85,B 0,C 180,E1 -9559.96,E2 -9559.96} C_VEL
LIN {X 0,Y 432.317,Z 76.134,A -85,B 0,C 180,E1 -9562.964,E2 -9562.964} C_VEL
LIN {X 0,Y 432.362,Z 76.117,A -85,B 0,C 180,E1 -9566.032,E2 -9566.032} C_VEL
LIN {X 0,Y 432.341,Z 76.128,A -85,B 0,C 180,E1 -9569.187,E2 -9569.187} C_VEL
LIN {X 0,Y 432.321,Z 76.132,A -85,B 0,C 180,E1 -9572.442,E2 -9572.442} C_VEL
LIN {X 0,Y 432.343,Z 76.124,A -85,B 0,C 180,E1 -9575.632,E2 -9575.632} C_VEL
LIN {X 0,Y 432.354,Z 76.129,A -85,B 0,C 180,E1 -9578.717,E2 -9578.717} C_VEL
LIN {X 0,Y 432.362,Z 76.121,A -85,B 0,C 180,E1 -9581.793,E2 -9581.793} C_VEL
LIN {X 0,Y 432.33,Z 76.133,A -85,B 0,C 180,E1 -9584.347,E2 -9584.347} C_VEL
LIN {X 0,Y 432.316,Z 76.107,A -85,B 0,C 180,E1 -9587.015,E2 -9587.015} C_VEL
LIN {X 0,Y 432.333,Z 76.118,A -85,B 0,C 180,E1 -9589.82,E2 -9589.82} C_VEL
LIN {X 0,Y 432.312,Z 76.13,A -85,B 0,C 180,E1 -9593.023,E2 -9593.023} C_VEL
LIN {X 0,Y 432.356,Z 76.111,A -85,B 0,C 180,E1 -9595.996,E2 -9595.996} C_VEL
LIN {X 0,Y 432.344,Z 76.128,A -85,B 0,C 180,E1 -9599.489,E2 -9599.489} C_VEL
LIN {X 0,Y 432.389,Z 76.124,A -85,B 0,C 180,E1 -9602.928,E2 -9602.928} C_VEL
LIN {X 0,Y 432.368,Z 76.13,A -85,B 0,C 180,E1 -9606.023,E2 -9606.023} C_VEL
LIN {X 0,Y 432.347,Z 76.131,A -85,B 0,C 180,E1 -9609.046,E2 -9609.046} C_VEL
LIN {X 0,Y 432.375,Z 76.129,A -85,B 0,C 180,E1 -9612.011,E2 -9612.011} C_VEL
LIN {X 0,Y 432.393,Z 76.126,A -85,B 0,C 180,E1 -9614.926,E2 -9614.926} C_VEL
LIN {X 0,Y 432.456,Z 76.119,A -85,B 0,C 180,E1 -9617.803,E2 -9617.803} C_VEL
LIN {X 0,Y 432.489,Z 76.115,A -85,B 0,C 180,E1 -9621.59,E2 -9621.59} C_VEL
LIN {X 0,Y 432.596,Z 76.101,A -85,B 0,C 180,E1 -9624.406,E2 -9624.406} C_VEL
LIN {X 0,Y 432.603,Z 76.099,A -85,B 0,C 180,E1 -9628.138,E2 -9628.138} C_VEL
LIN {X 0,Y 432.731,Z 76.084,A -85,B 0,C 180,E1 -9630,E2 -9630} C_VEL
LIN {X 0,Y 432.602,Z 76.1,A -85,B 0,C 180,E1 -9632.794,E2 -9632.794} C_VEL
LIN {X 0,Y 432.461,Z 76.116,A -85,B 0,C 180,E1 -9635.024,E2 -9635.024} C_VEL
LIN {X 0,Y 431.902,Z 76.187,A -85,B 0,C 180,E1 -9635.802,E2 -9635.802} C_VEL
LIN {X 0,Y 429.056,Z 76.543,A -85,B 0,C 180,E1 -9637.067,E2 -9637.067} C_VEL
LIN {X 0,Y 426.572,Z 76.852,A -85,B 0,C 180,E1 -9638.088,E2 -9638.088} C_VEL
LIN {X 0,Y 425.491,Z 76.987,A -85,B 0,C 180,E1 -9638.878,E2 -9638.878} C_VEL
LIN {X 0,Y 425.4,Z 76.996,A -85,B 0,C 180,E1 -9639.146,E2 -9639.146} C_VEL
LIN {X 0,Y 425.39,Z 76.999,A -85,B 0,C 180,E1 -9642.904,E2 -9642.904} C_VEL
LIN {X 0,Y 425.358,Z 77.003,A -85,B 0,C 180,E1 -9646.605,E2 -9646.605} C_VEL
LIN {X 0,Y 425.325,Z 77.005,A -85,B 0,C 180,E1 -9649.636,E2 -9649.636} C_VEL
LIN {X 0,Y 425.304,Z 77.007,A -85,B 0,C 180,E1 -9653.365,E2 -9653.365} C_VEL
LIN {X 0,Y 425.345,Z 77.002,A -85,B 0,C 180,E1 -9656.845,E2 -9656.845} C_VEL
LIN {X 0,Y 425.287,Z 76.996,A -85,B 0,C 180,E1 -9659.72,E2 -9659.72} C_VEL
LIN {X 0,Y 425.281,Z 77.006,A -85,B 0,C 180,E1 -9663.048,E2 -9663.048} C_VEL
LIN {X 0,Y 425.281,Z 76.997,A -85,B 0,C 180,E1 -9665.929,E2 -9665.929} C_VEL
LIN {X 0,Y 425.297,Z 77.006,A -85,B 0,C 180,E1 -9669.044,E2 -9669.044} C_VEL
LIN {X 0,Y 425.27,Z 76.983,A -85,B 0,C 180,E1 -9672.653,E2 -9672.653} C_VEL
LIN {X 0,Y 425.258,Z 77.012,A -85,B 0,C 180,E1 -9676.044,E2 -9676.044} C_VEL
LIN {X 0,Y 425.301,Z 77.001,A -85,B 0,C 180,E1 -9678.625,E2 -9678.625} C_VEL
LIN {X 0,Y 425.318,Z 77.003,A -85,B 0,C 180,E1 -9681.104,E2 -9681.104} C_VEL
LIN {X 0,Y 425.298,Z 77.003,A -85,B 0,C 180,E1 -9684.665,E2 -9684.665} C_VEL
LIN {X 0,Y 425.262,Z 77.009,A -85,B 0,C 180,E1 -9688.074,E2 -9688.074} C_VEL
LIN {X 0,Y 425.329,Z 76.993,A -85,B 0,C 180,E1 -9691.368,E2 -9691.368} C_VEL
LIN {X 0,Y 425.293,Z 77,A -85,B 0,C 180,E1 -9694.555,E2 -9694.555} C_VEL
LIN {X 0,Y 425.286,Z 77.005,A -85,B 0,C 180,E1 -9697.662,E2 -9697.662} C_VEL
LIN {X 0,Y 425.36,Z 76.983,A -85,B 0,C 180,E1 -9700.705,E2 -9700.705} C_VEL
LIN {X 0,Y 425.387,Z 76.99,A -85,B 0,C 180,E1 -9703.689,E2 -9703.689} C_VEL
LIN {X 0,Y 425.429,Z 76.985,A -85,B 0,C 180,E1 -9707.599,E2 -9707.599} C_VEL
LIN {X 0,Y 425.442,Z 76.973,A -85,B 0,C 180,E1 -9711.45,E2 -9711.45} C_VEL
LIN {X 0,Y 425.553,Z 76.979,A -85,B 0,C 180,E1 -9714.314,E2 -9714.314} C_VEL
LIN {X 0,Y 425.573,Z 76.961,A -85,B 0,C 180,E1 -9718.108,E2 -9718.108} C_VEL
LIN {X 0,Y 425.701,Z 76.937,A -85,B 0,C 180,E1 -9720.001,E2 -9720.001} C_VEL
LIN {X 0,Y 425.545,Z 76.971,A -85,B 0,C 180,E1 -9722.84,E2 -9722.84} C_VEL
LIN {X 0,Y 425.573,Z 76.976,A -85,B 0,C 180,E1 -9725.687,E2 -9725.687} C_VEL
LIN {X 0,Y 425.443,Z 76.972,A -85,B 0,C 180,E1 -9728.551,E2 -9728.551} C_VEL
LIN {X 0,Y 425.412,Z 76.986,A -85,B 0,C 180,E1 -9732.402,E2 -9732.402} C_VEL
LIN {X 0,Y 425.389,Z 76.987,A -85,B 0,C 180,E1 -9736.312,E2 -9736.312} C_VEL
LIN {X 0,Y 425.329,Z 76.989,A -85,B 0,C 180,E1 -9739.636,E2 -9739.636} C_VEL
LIN {X 0,Y 425.308,Z 77.007,A -85,B 0,C 180,E1 -9743.366,E2 -9743.366} C_VEL
LIN {X 0,Y 425.348,Z 76.987,A -85,B 0,C 180,E1 -9746.845,E2 -9746.845} C_VEL
LIN {X 0,Y 425.292,Z 77.006,A -85,B 0,C 180,E1 -9749.72,E2 -9749.72} C_VEL
LIN {X 0,Y 425.283,Z 77.001,A -85,B 0,C 180,E1 -9753.048,E2 -9753.048} C_VEL
LIN {X 0,Y 425.284,Z 77.004,A -85,B 0,C 180,E1 -9755.929,E2 -9755.929} C_VEL
LIN {X 0,Y 425.283,Z 77.004,A -85,B 0,C 180,E1 -9759.041,E2 -9759.041} C_VEL
LIN {X 0,Y 425.291,Z 77.006,A -85,B 0,C 180,E1 -9761.959,E2 -9761.959} C_VEL
LIN {X 0,Y 425.286,Z 77.005,A -85,B 0,C 180,E1 -9765.283,E2 -9765.283} C_VEL
LIN {X 0,Y 425.276,Z 76.999,A -85,B 0,C 180,E1 -9768.622,E2 -9768.622} C_VEL
LIN {X 0,Y 425.307,Z 77.001,A -85,B 0,C 180,E1 -9771.102,E2 -9771.102} C_VEL
LIN {X 0,Y 425.303,Z 76.997,A -85,B 0,C 180,E1 -9774.665,E2 -9774.665} C_VEL
LIN {X 0,Y 425.267,Z 77.006,A -85,B 0,C 180,E1 -9778.073,E2 -9778.073} C_VEL
LIN {X 0,Y 425.378,Z 77.169,A -85,B 0,C 180,E1 -9781.123,E2 -9781.123} C_VEL
LIN {X 0,Y 427.036,Z 86.047,A -85,B 0,C 180,E1 -9783.618,E2 -9783.618} C_VEL
LIN {X 0,Y 427.618,Z 91.08,A -85,B 0,C 180,E1 -9784.963,E2 -9784.963} C_VEL
LIN {X 0,Y 426.691,Z 105.578,A -85,B 0,C 180,E1 -9788.501,E2 -9788.501} C_VEL
LIN {X 0,Y 426.034,Z 115.475,A -85,B 0,C 180,E1 -9790.986,E2 -9790.986} C_VEL
LIN {X 0,Y 426.02,Z 116.782,A -85,B 0,C 180,E1 -9791.235,E2 -9791.235} C_VEL
LIN {X 0,Y 430.373,Z 141.379,A -85,B 0,C 180,E1 -9791.881,E2 -9791.881} C_VEL
LIN {X 0,Y 429.656,Z 221.383,A -85,B 0,C 180,E1 -9793.244,E2 -9793.244} C_VEL
LIN {X 0,Y 429.335,Z 231.279,A -85,B 0,C 180,E1 -9793.506,E2 -9793.506} C_VEL
LIN {X 0,Y 428.889,Z 241.254,A -85,B 0,C 180,E1 -9793.886,E2 -9793.886} C_VEL
LIN {X 0,Y 428.445,Z 250.611,A -85,B 0,C 180,E1 -9794.358,E2 -9794.358} C_VEL
LIN {X 0,Y 427.85,Z 260.753,A -85,B 0,C 180,E1 -9795.006,E2 -9795.006} C_VEL
LIN {X 0,Y 427.273,Z 269.75,A -85,B 0,C 180,E1 -9795.716,E2 -9795.716} C_VEL
LIN {X 0,Y 426.714,Z 278.119,A -85,B 0,C 180,E1 -9796.509,E2 -9796.509} C_VEL
LIN {X 0,Y 426.28,Z 285.878,A -85,B 0,C 180,E1 -9797.382,E2 -9797.382} C_VEL
LIN {X 0,Y 425.757,Z 293.098,A -85,B 0,C 180,E1 -9798.334,E2 -9798.334} C_VEL
LIN {X 0,Y 425.278,Z 299.298,A -85,B 0,C 180,E1 -9799.286,E2 -9799.286} C_VEL
LIN {X 0,Y 424.856,Z 305.836,A -85,B 0,C 180,E1 -9800.478,E2 -9800.478} C_VEL
LIN {X 0,Y 424.634,Z 310.338,A -85,B 0,C 180,E1 -9801.434,E2 -9801.434} C_VEL
LIN {X 0,Y 424.339,Z 315.828,A -85,B 0,C 180,E1 -9802.864,E2 -9802.864} C_VEL
LIN {X 0,Y 424.187,Z 320.151,A -85,B 0,C 180,E1 -9804.295,E2 -9804.295} C_VEL
LIN {X 0,Y 424.199,Z 322.518,A -85,B 0,C 180,E1 -9805.248,E2 -9805.248} C_VEL
LIN {X 0,Y 424.132,Z 325.701,A -85,B 0,C 180,E1 -9807.151,E2 -9807.151} C_VEL
LIN {X 0,Y 424.129,Z 326.757,A -85,B 0,C 180,E1 -9808.101,E2 -9808.101} C_VEL
LIN {X 0,Y 424.09,Z 327.344,A -85,B 0,C 180,E1 -9809.05,E2 -9809.05} C_VEL
LIN {X 0,Y 424.09,Z 327.344,A -85,B 0,C 180,E1 -9810.95,E2 -9810.95} C_VEL
LIN {X 0,Y 424.129,Z 326.757,A -85,B 0,C 180,E1 -9811.899,E2 -9811.899} C_VEL
LIN {X 0,Y 424.098,Z 324.314,A -85,B 0,C 180,E1 -9813.801,E2 -9813.801} C_VEL
LIN {X 0,Y 424.203,Z 321.369,A -85,B 0,C 180,E1 -9815.228,E2 -9815.228} C_VEL
LIN {X 0,Y 424.3,Z 317.382,A -85,B 0,C 180,E1 -9816.658,E2 -9816.658} C_VEL
LIN {X 0,Y 424.516,Z 312.254,A -85,B 0,C 180,E1 -9818.09,E2 -9818.09} C_VEL
LIN {X 0,Y 424.791,Z 306.992,A -85,B 0,C 180,E1 -9819.283,E2 -9819.283} C_VEL
LIN {X 0,Y 425.165,Z 300.674,A -85,B 0,C 180,E1 -9820.476,E2 -9820.476} C_VEL
LIN {X 0,Y 425.613,Z 294.724,A -85,B 0,C 180,E1 -9821.429,E2 -9821.429} C_VEL
LIN {X 0,Y 426.107,Z 287.797,A -85,B 0,C 180,E1 -9822.381,E2 -9822.381} C_VEL
LIN {X 0,Y 426.644,Z 279.615,A -85,B 0,C 180,E1 -9823.333,E2 -9823.333} C_VEL
LIN {X 0,Y 427.212,Z 270.824,A -85,B 0,C 180,E1 -9824.189,E2 -9824.189} C_VEL
LIN {X 0,Y 427.723,Z 262.384,A -85,B 0,C 180,E1 -9824.877,E2 -9824.877} C_VEL
LIN {X 0,Y 428.33,Z 252.625,A -85,B 0,C 180,E1 -9825.525,E2 -9825.525} C_VEL
LIN {X 0,Y 428.816,Z 243.831,A -85,B 0,C 180,E1 -9825.994,E2 -9825.994} C_VEL
LIN {X 0,Y 429.24,Z 233.902,A -85,B 0,C 180,E1 -9826.406,E2 -9826.406} C_VEL
LIN {X 0,Y 429.586,Z 224.046,A -85,B 0,C 180,E1 -9826.698,E2 -9826.698} C_VEL
LIN {X 0,Y 429.951,Z 199.241,A -85,B 0,C 180,E1 -9827.145,E2 -9827.145} C_VEL
LIN {X 0,Y 430.364,Z 141.111,A -85,B 0,C 180,E1 -9828.124,E2 -9828.124} C_VEL
LIN {X 0,Y 426.018,Z 116.772,A -85,B 0,C 180,E1 -9828.765,E2 -9828.765} C_VEL
LIN {X 0,Y 426.019,Z 115.475,A -85,B 0,C 180,E1 -9829.015,E2 -9829.015} C_VEL
LIN {X 0,Y 426.741,Z 104.7,A -85,B 0,C 180,E1 -9831.75,E2 -9831.75} C_VEL
LIN {X 0,Y 427.639,Z 91.444,A -85,B 0,C 180,E1 -9835.036,E2 -9835.036} C_VEL
LIN {X 0,Y 427.097,Z 86.187,A -85,B 0,C 180,E1 -9836.378,E2 -9836.378} C_VEL
LIN {X 0,Y 425.338,Z 77.08,A -85,B 0,C 180,E1 -9838.91,E2 -9838.91} C_VEL
LIN {X 0,Y 425.267,Z 77.007,A -85,B 0,C 180,E1 -9841.927,E2 -9841.927} C_VEL
LIN {X 0,Y 425.303,Z 76.998,A -85,B 0,C 180,E1 -9845.335,E2 -9845.335} C_VEL
LIN {X 0,Y 425.307,Z 77.002,A -85,B 0,C 180,E1 -9848.898,E2 -9848.898} C_VEL
LIN {X 0,Y 425.292,Z 77.008,A -85,B 0,C 180,E1 -9851.958,E2 -9851.958} C_VEL
LIN {X 0,Y 425.286,Z 77.006,A -85,B 0,C 180,E1 -9855.283,E2 -9855.283} C_VEL
LIN {X 0,Y 425.276,Z 77.008,A -85,B 0,C 180,E1 -9858.621,E2 -9858.621} C_VEL
LIN {X 0,Y 425.298,Z 77.004,A -85,B 0,C 180,E1 -9861.101,E2 -9861.101} C_VEL
LIN {X 0,Y 425.301,Z 77.004,A -85,B 0,C 180,E1 -9864.664,E2 -9864.664} C_VEL
LIN {X 0,Y 425.266,Z 77.008,A -85,B 0,C 180,E1 -9868.073,E2 -9868.073} C_VEL
LIN {X 0,Y 425.332,Z 76.994,A -85,B 0,C 180,E1 -9871.367,E2 -9871.367} C_VEL
LIN {X 0,Y 425.296,Z 76.998,A -85,B 0,C 180,E1 -9874.554,E2 -9874.554} C_VEL
LIN {X 0,Y 425.289,Z 77.004,A -85,B 0,C 180,E1 -9877.661,E2 -9877.661} C_VEL
LIN {X 0,Y 425.363,Z 76.981,A -85,B 0,C 180,E1 -9880.704,E2 -9880.704} C_VEL
LIN {X 0,Y 425.389,Z 76.987,A -85,B 0,C 180,E1 -9883.688,E2 -9883.688} C_VEL
LIN {X 0,Y 425.412,Z 76.986,A -85,B 0,C 180,E1 -9887.598,E2 -9887.598} C_VEL
LIN {X 0,Y 425.443,Z 76.972,A -85,B 0,C 180,E1 -9891.449,E2 -9891.449} C_VEL
LIN {X 0,Y 425.573,Z 76.976,A -85,B 0,C 180,E1 -9894.313,E2 -9894.313} C_VEL
LIN {X 0,Y 425.573,Z 76.962,A -85,B 0,C 180,E1 -9898.107,E2 -9898.107} C_VEL
LIN {X 0,Y 425.701,Z 76.937,A -85,B 0,C 180,E1 -9899.999,E2 -9899.999} C_VEL
LIN {X 0,Y 425.545,Z 76.969,A -85,B 0,C 180,E1 -9902.839,E2 -9902.839} C_VEL
LIN {X 0,Y 425.53,Z 76.973,A -85,B 0,C 180,E1 -9906.638,E2 -9906.638} C_VEL
LIN {X 0,Y 425.402,Z 76.976,A -85,B 0,C 180,E1 -9909.509,E2 -9909.509} C_VEL
LIN {X 0,Y 425.403,Z 76.989,A -85,B 0,C 180,E1 -9912.91,E2 -9912.91} C_VEL
LIN {X 0,Y 425.36,Z 76.994,A -85,B 0,C 180,E1 -9916.605,E2 -9916.605} C_VEL
LIN {X 0,Y 425.327,Z 76.99,A -85,B 0,C 180,E1 -9919.635,E2 -9919.635} C_VEL
LIN {X 0,Y 425.305,Z 77.009,A -85,B 0,C 180,E1 -9923.365,E2 -9923.365} C_VEL
LIN {X 0,Y 425.346,Z 76.989,A -85,B 0,C 180,E1 -9926.844,E2 -9926.844} C_VEL
LIN {X 0,Y 425.289,Z 77.006,A -85,B 0,C 180,E1 -9929.719,E2 -9929.719} C_VEL
LIN {X 0,Y 425.279,Z 77.004,A -85,B 0,C 180,E1 -9933.048,E2 -9933.048} C_VEL
LIN {X 0,Y 425.282,Z 77.003,A -85,B 0,C 180,E1 -9935.929,E2 -9935.929} C_VEL
LIN {X 0,Y 425.307,Z 77.003,A -85,B 0,C 180,E1 -9939.045,E2 -9939.045} C_VEL
LIN {X 0,Y 425.312,Z 77,A -85,B 0,C 180,E1 -9941.962,E2 -9941.962} C_VEL
LIN {X 0,Y 425.281,Z 77.001,A -85,B 0,C 180,E1 -9945.283,E2 -9945.283} C_VEL
LIN {X 0,Y 425.27,Z 76.984,A -85,B 0,C 180,E1 -9948.621,E2 -9948.621} C_VEL
LIN {X 0,Y 425.31,Z 77.004,A -85,B 0,C 180,E1 -9951.103,E2 -9951.103} C_VEL
LIN {X 0,Y 425.297,Z 76.989,A -85,B 0,C 180,E1 -9954.664,E2 -9954.664} C_VEL
LIN {X 0,Y 425.262,Z 77.016,A -85,B 0,C 180,E1 -9958.073,E2 -9958.073} C_VEL
LIN {X 0,Y 425.328,Z 76.993,A -85,B 0,C 180,E1 -9961.368,E2 -9961.368} C_VEL
LIN {X 0,Y 425.292,Z 77.009,A -85,B 0,C 180,E1 -9964.555,E2 -9964.555} C_VEL
LIN {X 0,Y 425.284,Z 77.013,A -85,B 0,C 180,E1 -9967.661,E2 -9967.661} C_VEL
LIN {X 0,Y 425.359,Z 77.001,A -85,B 0,C 180,E1 -9970.704,E2 -9970.704} C_VEL
LIN {X 0,Y 425.385,Z 77.001,A -85,B 0,C 180,E1 -9973.688,E2 -9973.688} C_VEL
LIN {X 0,Y 425.409,Z 76.997,A -85,B 0,C 180,E1 -9977.598,E2 -9977.598} C_VEL
LIN {X 0,Y 425.439,Z 76.993,A -85,B 0,C 180,E1 -9981.45,E2 -9981.45} C_VEL
LIN {X 0,Y 425.552,Z 76.978,A -85,B 0,C 180,E1 -9984.313,E2 -9984.313} C_VEL
LIN {X 0,Y 425.572,Z 76.975,A -85,B 0,C 180,E1 -9988.107,E2 -9988.107} C_VEL
LIN {X 0,Y 425.7,Z 76.96,A -85,B 0,C 180,E1 -9990,E2 -9990} C_VEL
LIN {X 0,Y 425.553,Z 76.978,A -85,B 0,C 180,E1 -9992.84,E2 -9992.84} C_VEL
LIN {X 0,Y 425.528,Z 76.982,A -85,B 0,C 180,E1 -9996.639,E2 -9996.639} C_VEL
LIN {X 0,Y 425.4,Z 76.996,A -85,B 0,C 180,E1 -9999.146,E2 -9999.146} C_VEL
LIN {X 0,Y 424.727,Z 77.081,A -85,B 0,C 180,E1 -9999.936,E2 -9999.936} C_VEL
LIN {X 0,Y 421.879,Z 77.437,A -85,B 0,C 180,E1 -10001.219,E2 -10001.219} C_VEL
LIN {X 0,Y 419.464,Z 77.737,A -85,B 0,C 180,E1 -10002.256,E2 -10002.256} C_VEL
LIN {X 0,Y 418.413,Z 77.868,A -85,B 0,C 180,E1 -10003.056,E2 -10003.056} C_VEL
LIN {X 0,Y 418.319,Z 77.878,A -85,B 0,C 180,E1 -10003.328,E2 -10003.328} C_VEL
LIN {X 0,Y 418.309,Z 77.881,A -85,B 0,C 180,E1 -10006.736,E2 -10006.736} C_VEL
LIN {X 0,Y 418.267,Z 77.885,A -85,B 0,C 180,E1 -10009.791,E2 -10009.791} C_VEL
LIN {X 0,Y 418.235,Z 77.89,A -85,B 0,C 180,E1 -10012.736,E2 -10012.736} C_VEL
LIN {X 0,Y 418.267,Z 77.887,A -85,B 0,C 180,E1 -10015.904,E2 -10015.904} C_VEL
LIN {X 0,Y 418.261,Z 77.87,A -85,B 0,C 180,E1 -10019.162,E2 -10019.162} C_VEL
LIN {X 0,Y 418.257,Z 77.88,A -85,B 0,C 180,E1 -10022.845,E2 -10022.845} C_VEL
LIN {X 0,Y 418.245,Z 77.879,A -85,B 0,C 180,E1 -10026.239,E2 -10026.239} C_VEL
LIN {X 0,Y 418.248,Z 77.877,A -85,B 0,C 180,E1 -10029.682,E2 -10029.682} C_VEL
LIN {X 0,Y 418.225,Z 77.857,A -85,B 0,C 180,E1 -10032.321,E2 -10032.321} C_VEL
LIN {X 0,Y 418.232,Z 77.881,A -85,B 0,C 180,E1 -10035.109,E2 -10035.109} C_VEL
LIN {X 0,Y 418.253,Z 77.882,A -85,B 0,C 180,E1 -10037.769,E2 -10037.769} C_VEL
LIN {X 0,Y 418.263,Z 77.878,A -85,B 0,C 180,E1 -10040.617,E2 -10040.617} C_VEL
LIN {X 0,Y 418.243,Z 77.88,A -85,B 0,C 180,E1 -10043.977,E2 -10043.977} C_VEL
LIN {X 0,Y 418.255,Z 77.881,A -85,B 0,C 180,E1 -10047.156,E2 -10047.156} C_VEL
LIN {X 0,Y 418.266,Z 77.879,A -85,B 0,C 180,E1 -10050.896,E2 -10050.896} C_VEL
LIN {X 0,Y 418.269,Z 77.872,A -85,B 0,C 180,E1 -10054.096,E2 -10054.096} C_VEL
LIN {X 0,Y 418.236,Z 77.885,A -85,B 0,C 180,E1 -10057.264,E2 -10057.264} C_VEL
LIN {X 0,Y 418.281,Z 77.866,A -85,B 0,C 180,E1 -10060.365,E2 -10060.365} C_VEL
LIN {X 0,Y 418.316,Z 77.871,A -85,B 0,C 180,E1 -10063.405,E2 -10063.405} C_VEL
LIN {X 0,Y 418.354,Z 77.867,A -85,B 0,C 180,E1 -10066.994,E2 -10066.994} C_VEL
LIN {X 0,Y 418.343,Z 77.853,A -85,B 0,C 180,E1 -10070.329,E2 -10070.329} C_VEL
LIN {X 0,Y 418.493,Z 77.849,A -85,B 0,C 180,E1 -10073.25,E2 -10073.25} C_VEL
LIN {X 0,Y 418.338,Z 77.872,A -85,B 0,C 180,E1 -10075.182,E2 -10075.182} C_VEL
LIN {X 0,Y 418.542,Z 77.837,A -85,B 0,C 180,E1 -10078.076,E2 -10078.076} C_VEL
LIN {X 0,Y 418.67,Z 77.812,A -85,B 0,C 180,E1 -10080.001,E2 -10080.001} C_VEL
LIN {X 0,Y 418.5,Z 77.848,A -85,B 0,C 180,E1 -10082.888,E2 -10082.888} C_VEL
LIN {X 0,Y 418.529,Z 77.852,A -85,B 0,C 180,E1 -10085.783,E2 -10085.783} C_VEL
LIN {X 0,Y 418.4,Z 77.848,A -85,B 0,C 180,E1 -10088.696,E2 -10088.696} C_VEL
LIN {X 0,Y 418.315,Z 77.865,A -85,B 0,C 180,E1 -10091.632,E2 -10091.632} C_VEL
LIN {X 0,Y 418.303,Z 77.875,A -85,B 0,C 180,E1 -10094.597,E2 -10094.597} C_VEL
LIN {X 0,Y 418.288,Z 77.864,A -85,B 0,C 180,E1 -10097.604,E2 -10097.604} C_VEL
LIN {X 0,Y 418.251,Z 77.874,A -85,B 0,C 180,E1 -10100.663,E2 -10100.663} C_VEL
LIN {X 0,Y 418.289,Z 77.877,A -85,B 0,C 180,E1 -10103.782,E2 -10103.782} C_VEL
LIN {X 0,Y 418.311,Z 77.863,A -85,B 0,C 180,E1 -10107.071,E2 -10107.071} C_VEL
LIN {X 0,Y 418.246,Z 77.883,A -85,B 0,C 180,E1 -10110.273,E2 -10110.273} C_VEL
LIN {X 0,Y 418.25,Z 77.871,A -85,B 0,C 180,E1 -10113.678,E2 -10113.678} C_VEL
LIN {X 0,Y 418.241,Z 77.887,A -85,B 0,C 180,E1 -10117.225,E2 -10117.225} C_VEL
LIN {X 0,Y 418.246,Z 77.876,A -85,B 0,C 180,E1 -10119.683,E2 -10119.683} C_VEL
LIN {X 0,Y 418.231,Z 77.888,A -85,B 0,C 180,E1 -10122.322,E2 -10122.322} C_VEL
LIN {X 0,Y 418.237,Z 77.884,A -85,B 0,C 180,E1 -10125.109,E2 -10125.109} C_VEL
LIN {X 0,Y 418.242,Z 77.884,A -85,B 0,C 180,E1 -10127.767,E2 -10127.767} C_VEL
LIN {X 0,Y 418.257,Z 77.88,A -85,B 0,C 180,E1 -10131.559,E2 -10131.559} C_VEL
LIN {X 0,Y 418.262,Z 77.876,A -85,B 0,C 180,E1 -10135.159,E2 -10135.159} C_VEL
LIN {X 0,Y 418.248,Z 77.882,A -85,B 0,C 180,E1 -10137.472,E2 -10137.472} C_VEL
LIN {X 0,Y 418.324,Z 78.086,A -85,B 0,C 180,E1 -10140.883,E2 -10140.883} C_VEL
LIN {X 0,Y 419.87,Z 85.909,A -85,B 0,C 180,E1 -10143.132,E2 -10143.132} C_VEL
LIN {X 0,Y 420.65,Z 92.387,A -85,B 0,C 180,E1 -10144.895,E2 -10144.895} C_VEL
LIN {X 0,Y 419.718,Z 106.449,A -85,B 0,C 180,E1 -10148.384,E2 -10148.384} C_VEL
LIN {X 0,Y 419.042,Z 116.316,A -85,B 0,C 180,E1 -10150.879,E2 -10150.879} C_VEL
LIN {X 0,Y 419.589,Z 119.667,A -85,B 0,C 180,E1 -10151.019,E2 -10151.019} C_VEL
LIN {X 0,Y 423.653,Z 142.325,A -85,B 0,C 180,E1 -10151.603,E2 -10151.603} C_VEL
LIN {X 0,Y 422.863,Z 221.192,A -85,B 0,C 180,E1 -10152.967,E2 -10152.967} C_VEL
LIN {X 0,Y 422.514,Z 231.963,A -85,B 0,C 180,E1 -10153.263,E2 -10153.263} C_VEL
LIN {X 0,Y 422.067,Z 241.063,A -85,B 0,C 180,E1 -10153.618,E2 -10153.618} C_VEL
LIN {X 0,Y 421.617,Z 250.421,A -85,B 0,C 180,E1 -10154.098,E2 -10154.098} C_VEL
LIN {X 0,Y 420.964,Z 260.561,A -85,B 0,C 180,E1 -10154.755,E2 -10154.755} C_VEL
LIN {X 0,Y 420.39,Z 269.559,A -85,B 0,C 180,E1 -10155.477,E2 -10155.477} C_VEL
LIN {X 0,Y 419.773,Z 277.943,A -85,B 0,C 180,E1 -10156.283,E2 -10156.283} C_VEL
LIN {X 0,Y 419.324,Z 285.687,A -85,B 0,C 180,E1 -10157.169,E2 -10157.169} C_VEL
LIN {X 0,Y 418.783,Z 292.907,A -85,B 0,C 180,E1 -10158.137,E2 -10158.137} C_VEL
LIN {X 0,Y 418.283,Z 299.107,A -85,B 0,C 180,E1 -10159.104,E2 -10159.104} C_VEL
LIN {X 0,Y 417.816,Z 305.644,A -85,B 0,C 180,E1 -10160.316,E2 -10160.316} C_VEL
LIN {X 0,Y 417.57,Z 310.147,A -85,B 0,C 180,E1 -10161.288,E2 -10161.288} C_VEL
LIN {X 0,Y 417.265,Z 315.637,A -85,B 0,C 180,E1 -10162.743,E2 -10162.743} C_VEL
LIN {X 0,Y 417.104,Z 319.96,A -85,B 0,C 180,E1 -10164.198,E2 -10164.198} C_VEL
LIN {X 0,Y 417.105,Z 322.327,A -85,B 0,C 180,E1 -10165.167,E2 -10165.167} C_VEL
LIN {X 0,Y 417.028,Z 325.51,A -85,B 0,C 180,E1 -10167.102,E2 -10167.102} C_VEL
LIN {X 0,Y 417.057,Z 326.568,A -85,B 0,C 180,E1 -10168.069,E2 -10168.069} C_VEL
LIN {X 0,Y 417.012,Z 327.154,A -85,B 0,C 180,E1 -10169.034,E2 -10169.034} C_VEL
LIN {X 0,Y 417.012,Z 327.154,A -85,B 0,C 180,E1 -10170.966,E2 -10170.966} C_VEL
LIN {X 0,Y 417.057,Z 326.568,A -85,B 0,C 180,E1 -10171.931,E2 -10171.931} C_VEL
LIN {X 0,Y 417.014,Z 324.123,A -85,B 0,C 180,E1 -10173.865,E2 -10173.865} C_VEL
LIN {X 0,Y 417.118,Z 321.178,A -85,B 0,C 180,E1 -10175.317,E2 -10175.317} C_VEL
LIN {X 0,Y 417.232,Z 317.191,A -85,B 0,C 180,E1 -10176.771,E2 -10176.771} C_VEL
LIN {X 0,Y 417.457,Z 312.062,A -85,B 0,C 180,E1 -10178.227,E2 -10178.227} C_VEL
LIN {X 0,Y 417.755,Z 306.8,A -85,B 0,C 180,E1 -10179.441,E2 -10179.441} C_VEL
LIN {X 0,Y 418.145,Z 300.483,A -85,B 0,C 180,E1 -10180.654,E2 -10180.654} C_VEL
LIN {X 0,Y 418.64,Z 294.533,A -85,B 0,C 180,E1 -10181.622,E2 -10181.622} C_VEL
LIN {X 0,Y 419.143,Z 287.605,A -85,B 0,C 180,E1 -10182.59,E2 -10182.59} C_VEL
LIN {X 0,Y 419.723,Z 279.424,A -85,B 0,C 180,E1 -10183.557,E2 -10183.557} C_VEL
LIN {X 0,Y 420.298,Z 270.755,A -85,B 0,C 180,E1 -10184.417,E2 -10184.417} C_VEL
LIN {X 0,Y 420.862,Z 262.193,A -85,B 0,C 180,E1 -10185.125,E2 -10185.125} C_VEL
LIN {X 0,Y 421.488,Z 252.435,A -85,B 0,C 180,E1 -10185.783,E2 -10185.783} C_VEL
LIN {X 0,Y 422.038,Z 242.352,A -85,B 0,C 180,E1 -10186.321,E2 -10186.321} C_VEL
LIN {X 0,Y 422.481,Z 232.837,A -85,B 0,C 180,E1 -10186.707,E2 -10186.707} C_VEL
LIN {X 0,Y 422.822,Z 222.524,A -85,B 0,C 180,E1 -10187.004,E2 -10187.004} C_VEL
LIN {X 0,Y 423.504,Z 163.224,A -85,B 0,C 180,E1 -10188.039,E2 -10188.039} C_VEL
LIN {X 0,Y 423.66,Z 142.145,A -85,B 0,C 180,E1 -10188.4,E2 -10188.4} C_VEL
LIN {X 0,Y 419.053,Z 116.84,A -85,B 0,C 180,E1 -10189.071,E2 -10189.071} C_VEL
LIN {X 0,Y 419.025,Z 115.783,A -85,B 0,C 180,E1 -10189.217,E2 -10189.217} C_VEL
LIN {X 0,Y 419.812,Z 104.522,A -85,B 0,C 180,E1 -10192.127,E2 -10192.127} C_VEL
LIN {X 0,Y 420.684,Z 92.675,A -85,B 0,C 180,E1 -10195.119,E2 -10195.119} C_VEL
LIN {X 0,Y 420.077,Z 87.1,A -85,B 0,C 180,E1 -10196.586,E2 -10196.586} C_VEL
LIN {X 0,Y 418.279,Z 77.968,A -85,B 0,C 180,E1 -10199.161,E2 -10199.161} C_VEL
LIN {X 0,Y 418.26,Z 77.883,A -85,B 0,C 180,E1 -10202.844,E2 -10202.844} C_VEL
LIN {X 0,Y 418.251,Z 77.882,A -85,B 0,C 180,E1 -10206.238,E2 -10206.238} C_VEL
LIN {X 0,Y 418.249,Z 77.869,A -85,B 0,C 180,E1 -10209.682,E2 -10209.682} C_VEL
LIN {X 0,Y 418.232,Z 77.886,A -85,B 0,C 180,E1 -10212.321,E2 -10212.321} C_VEL
LIN {X 0,Y 418.237,Z 77.884,A -85,B 0,C 180,E1 -10215.108,E2 -10215.108} C_VEL
LIN {X 0,Y 418.241,Z 77.886,A -85,B 0,C 180,E1 -10217.766,E2 -10217.766} C_VEL
LIN {X 0,Y 418.247,Z 77.877,A -85,B 0,C 180,E1 -10220.62,E2 -10220.62} C_VEL
LIN {X 0,Y 418.244,Z 77.881,A -85,B 0,C 180,E1 -10223.975,E2 -10223.975} C_VEL
LIN {X 0,Y 418.259,Z 77.879,A -85,B 0,C 180,E1 -10227.156,E2 -10227.156} C_VEL
LIN {X 0,Y 418.27,Z 77.879,A -85,B 0,C 180,E1 -10230.895,E2 -10230.895} C_VEL
LIN {X 0,Y 418.272,Z 77.869,A -85,B 0,C 180,E1 -10234.096,E2 -10234.096} C_VEL
LIN {X 0,Y 418.239,Z 77.884,A -85,B 0,C 180,E1 -10237.263,E2 -10237.263} C_VEL
LIN {X 0,Y 418.284,Z 77.865,A -85,B 0,C 180,E1 -10240.364,E2 -10240.364} C_VEL
LIN {X 0,Y 418.318,Z 77.868,A -85,B 0,C 180,E1 -10243.404,E2 -10243.404} C_VEL
LIN {X 0,Y 418.347,Z 77.867,A -85,B 0,C 180,E1 -10246.999,E2 -10246.999} C_VEL
LIN {X 0,Y 418.341,Z 77.853,A -85,B 0,C 180,E1 -10250.328,E2 -10250.328} C_VEL
LIN {X 0,Y 418.513,Z 77.842,A -85,B 0,C 180,E1 -10252.279,E2 -10252.279} C_VEL
LIN {X 0,Y 418.529,Z 77.852,A -85,B 0,C 180,E1 -10254.217,E2 -10254.217} C_VEL
LIN {X 0,Y 418.542,Z 77.838,A -85,B 0,C 180,E1 -10258.075,E2 -10258.075} C_VEL
LIN {X 0,Y 418.67,Z 77.812,A -85,B 0,C 180,E1 -10259.999,E2 -10259.999} C_VEL
LIN {X 0,Y 418.5,Z 77.847,A -85,B 0,C 180,E1 -10262.887,E2 -10262.887} C_VEL
LIN {X 0,Y 418.493,Z 77.849,A -85,B 0,C 180,E1 -10266.75,E2 -10266.75} C_VEL
LIN {X 0,Y 418.343,Z 77.853,A -85,B 0,C 180,E1 -10269.671,E2 -10269.671} C_VEL
LIN {X 0,Y 418.354,Z 77.867,A -85,B 0,C 180,E1 -10273.006,E2 -10273.006} C_VEL
LIN {X 0,Y 418.312,Z 77.872,A -85,B 0,C 180,E1 -10276.735,E2 -10276.735} C_VEL
LIN {X 0,Y 418.269,Z 77.869,A -85,B 0,C 180,E1 -10279.79,E2 -10279.79} C_VEL
LIN {X 0,Y 418.236,Z 77.885,A -85,B 0,C 180,E1 -10282.736,E2 -10282.736} C_VEL
LIN {X 0,Y 418.269,Z 77.872,A -85,B 0,C 180,E1 -10285.904,E2 -10285.904} C_VEL
LIN {X 0,Y 418.262,Z 77.881,A -85,B 0,C 180,E1 -10289.161,E2 -10289.161} C_VEL
LIN {X 0,Y 418.255,Z 77.881,A -85,B 0,C 180,E1 -10292.844,E2 -10292.844} C_VEL
LIN {X 0,Y 418.246,Z 77.881,A -85,B 0,C 180,E1 -10296.238,E2 -10296.238} C_VEL
LIN {X 0,Y 418.261,Z 77.877,A -85,B 0,C 180,E1 -10299.68,E2 -10299.68} C_VEL
LIN {X 0,Y 418.242,Z 77.884,A -85,B 0,C 180,E1 -10302.323,E2 -10302.323} C_VEL
LIN {X 0,Y 418.232,Z 77.879,A -85,B 0,C 180,E1 -10305.108,E2 -10305.108} C_VEL
LIN {X 0,Y 418.236,Z 77.856,A -85,B 0,C 180,E1 -10307.766,E2 -10307.766} C_VEL
LIN {X 0,Y 418.254,Z 77.882,A -85,B 0,C 180,E1 -10310.618,E2 -10310.618} C_VEL
LIN {X 0,Y 418.243,Z 77.876,A -85,B 0,C 180,E1 -10313.976,E2 -10313.976} C_VEL
LIN {X 0,Y 418.254,Z 77.881,A -85,B 0,C 180,E1 -10317.156,E2 -10317.156} C_VEL
LIN {X 0,Y 418.265,Z 77.869,A -85,B 0,C 180,E1 -10320.895,E2 -10320.895} C_VEL
LIN {X 0,Y 418.267,Z 77.887,A -85,B 0,C 180,E1 -10324.096,E2 -10324.096} C_VEL
LIN {X 0,Y 418.235,Z 77.89,A -85,B 0,C 180,E1 -10327.264,E2 -10327.264} C_VEL
LIN {X 0,Y 418.28,Z 77.883,A -85,B 0,C 180,E1 -10330.364,E2 -10330.364} C_VEL
LIN {X 0,Y 418.314,Z 77.881,A -85,B 0,C 180,E1 -10333.405,E2 -10333.405} C_VEL
LIN {X 0,Y 418.343,Z 77.877,A -85,B 0,C 180,E1 -10336.999,E2 -10336.999} C_VEL
LIN {X 0,Y 418.338,Z 77.877,A -85,B 0,C 180,E1 -10340.329,E2 -10340.329} C_VEL
LIN {X 0,Y 418.491,Z 77.858,A -85,B 0,C 180,E1 -10343.249,E2 -10343.249} C_VEL
LIN {X 0,Y 418.338,Z 77.878,A -85,B 0,C 180,E1 -10345.182,E2 -10345.182} C_VEL
LIN {X 0,Y 418.541,Z 77.851,A -85,B 0,C 180,E1 -10348.075,E2 -10348.075} C_VEL
LIN {X 0,Y 418.67,Z 77.836,A -85,B 0,C 180,E1 -10350,E2 -10350} C_VEL
LIN {X 0,Y 418.507,Z 77.856,A -85,B 0,C 180,E1 -10352.888,E2 -10352.888} C_VEL
LIN {X 0,Y 418.491,Z 77.858,A -85,B 0,C 180,E1 -10356.751,E2 -10356.751} C_VEL
LIN {X 0,Y 418.338,Z 77.877,A -85,B 0,C 180,E1 -10359.671,E2 -10359.671} C_VEL
LIN {X 0,Y 418.319,Z 77.878,A -85,B 0,C 180,E1 -10363.328,E2 -10363.328} C_VEL
LIN {X 0,Y 417.626,Z 77.967,A -85,B 0,C 180,E1 -10364.131,E2 -10364.131} C_VEL
LIN {X 0,Y 414.748,Z 78.324,A -85,B 0,C 180,E1 -10365.436,E2 -10365.436} C_VEL
LIN {X 0,Y 412.335,Z 78.625,A -85,B 0,C 180,E1 -10366.491,E2 -10366.491} C_VEL
LIN {X 0,Y 411.313,Z 78.751,A -85,B 0,C 180,E1 -10367.306,E2 -10367.306} C_VEL
LIN {X 0,Y 411.236,Z 78.76,A -85,B 0,C 180,E1 -10367.582,E2 -10367.582} C_VEL
LIN {X 0,Y 411.193,Z 78.766,A -85,B 0,C 180,E1 -10371.034,E2 -10371.034} C_VEL
LIN {X 0,Y 411.224,Z 78.764,A -85,B 0,C 180,E1 -10374.215,E2 -10374.215} C_VEL
LIN {X 0,Y 411.255,Z 78.758,A -85,B 0,C 180,E1 -10377.478,E2 -10377.478} C_VEL
LIN {X 0,Y 411.187,Z 78.763,A -85,B 0,C 180,E1 -10380.848,E2 -10380.848} C_VEL
LIN {X 0,Y 411.203,Z 78.738,A -85,B 0,C 180,E1 -10384.334,E2 -10384.334} C_VEL
LIN {X 0,Y 411.197,Z 78.767,A -85,B 0,C 180,E1 -10387.973,E2 -10387.973} C_VEL
LIN {X 0,Y 411.178,Z 78.75,A -85,B 0,C 180,E1 -10390.504,E2 -10390.504} C_VEL
LIN {X 0,Y 411.169,Z 78.74,A -85,B 0,C 180,E1 -10393.134,E2 -10393.134} C_VEL
LIN {X 0,Y 411.164,Z 78.769,A -85,B 0,C 180,E1 -10395.881,E2 -10395.881} C_VEL
LIN {X 0,Y 411.197,Z 78.758,A -85,B 0,C 180,E1 -10398.766,E2 -10398.766} C_VEL
LIN {X 0,Y 411.201,Z 78.763,A -85,B 0,C 180,E1 -10402.028,E2 -10402.028} C_VEL
LIN {X 0,Y 411.203,Z 78.752,A -85,B 0,C 180,E1 -10405.667,E2 -10405.667} C_VEL
LIN {X 0,Y 411.187,Z 78.768,A -85,B 0,C 180,E1 -10409.153,E2 -10409.153} C_VEL
LIN {X 0,Y 411.257,Z 78.742,A -85,B 0,C 180,E1 -10412.523,E2 -10412.523} C_VEL
LIN {X 0,Y 411.225,Z 78.757,A -85,B 0,C 180,E1 -10415.785,E2 -10415.785} C_VEL
LIN {X 0,Y 411.195,Z 78.755,A -85,B 0,C 180,E1 -10418.966,E2 -10418.966} C_VEL
LIN {X 0,Y 411.251,Z 78.74,A -85,B 0,C 180,E1 -10422.085,E2 -10422.085} C_VEL
LIN {X 0,Y 411.261,Z 78.755,A -85,B 0,C 180,E1 -10425.148,E2 -10425.148} C_VEL
LIN {X 0,Y 411.297,Z 78.743,A -85,B 0,C 180,E1 -10428.168,E2 -10428.168} C_VEL
LIN {X 0,Y 411.481,Z 78.717,A -85,B 0,C 180,E1 -10432.147,E2 -10432.147} C_VEL
LIN {X 0,Y 411.475,Z 78.729,A -85,B 0,C 180,E1 -10434.119,E2 -10434.119} C_VEL
LIN {X 0,Y 411.511,Z 78.713,A -85,B 0,C 180,E1 -10438.043,E2 -10438.043} C_VEL
LIN {X 0,Y 411.64,Z 78.686,A -85,B 0,C 180,E1 -10440.001,E2 -10440.001} C_VEL
LIN {X 0,Y 411.457,Z 78.725,A -85,B 0,C 180,E1 -10442.938,E2 -10442.938} C_VEL
LIN {X 0,Y 411.489,Z 78.728,A -85,B 0,C 180,E1 -10445.882,E2 -10445.882} C_VEL
LIN {X 0,Y 411.482,Z 78.716,A -85,B 0,C 180,E1 -10447.854,E2 -10447.854} C_VEL
LIN {X 0,Y 411.284,Z 78.744,A -85,B 0,C 180,E1 -10451.833,E2 -10451.833} C_VEL
LIN {X 0,Y 411.261,Z 78.753,A -85,B 0,C 180,E1 -10454.853,E2 -10454.853} C_VEL
LIN {X 0,Y 411.253,Z 78.736,A -85,B 0,C 180,E1 -10457.916,E2 -10457.916} C_VEL
LIN {X 0,Y 411.197,Z 78.755,A -85,B 0,C 180,E1 -10461.035,E2 -10461.035} C_VEL
LIN {X 0,Y 411.228,Z 78.755,A -85,B 0,C 180,E1 -10464.216,E2 -10464.216} C_VEL
LIN {X 0,Y 411.26,Z 78.742,A -85,B 0,C 180,E1 -10467.478,E2 -10467.478} C_VEL
LIN {X 0,Y 411.19,Z 78.767,A -85,B 0,C 180,E1 -10470.848,E2 -10470.848} C_VEL
LIN {X 0,Y 411.207,Z 78.748,A -85,B 0,C 180,E1 -10474.334,E2 -10474.334} C_VEL
LIN {X 0,Y 411.193,Z 78.763,A -85,B 0,C 180,E1 -10477.974,E2 -10477.974} C_VEL
LIN {X 0,Y 411.165,Z 78.767,A -85,B 0,C 180,E1 -10481.229,E2 -10481.229} C_VEL
LIN {X 0,Y 411.177,Z 78.763,A -85,B 0,C 180,E1 -10484.491,E2 -10484.491} C_VEL
LIN {X 0,Y 411.179,Z 78.761,A -85,B 0,C 180,E1 -10488.195,E2 -10488.195} C_VEL
LIN {X 0,Y 411.218,Z 78.749,A -85,B 0,C 180,E1 -10490.776,E2 -10490.776} C_VEL
LIN {X 0,Y 411.202,Z 78.753,A -85,B 0,C 180,E1 -10494.472,E2 -10494.472} C_VEL
LIN {X 0,Y 411.21,Z 78.762,A -85,B 0,C 180,E1 -10496.874,E2 -10496.874} C_VEL
LIN {X 0,Y 411.259,Z 78.867,A -85,B 0,C 180,E1 -10500.576,E2 -10500.576} C_VEL
LIN {X 0,Y 412.995,Z 87.705,A -85,B 0,C 180,E1 -10503.195,E2 -10503.195} C_VEL
LIN {X 0,Y 413.678,Z 93.858,A -85,B 0,C 180,E1 -10504.867,E2 -10504.867} C_VEL
LIN {X 0,Y 412.739,Z 107.32,A -85,B 0,C 180,E1 -10508.263,E2 -10508.263} C_VEL
LIN {X 0,Y 412.084,Z 116.126,A -85,B 0,C 180,E1 -10510.543,E2 -10510.543} C_VEL
LIN {X 0,Y 412.536,Z 118.841,A -85,B 0,C 180,E1 -10510.671,E2 -10510.671} C_VEL
LIN {X 0,Y 416.972,Z 143.561,A -85,B 0,C 180,E1 -10511.323,E2 -10511.323} C_VEL
LIN {X 0,Y 416.097,Z 221.002,A -85,B 0,C 180,E1 -10512.681,E2 -10512.681} C_VEL
LIN {X 0,Y 415.773,Z 230.899,A -85,B 0,C 180,E1 -10512.952,E2 -10512.952} C_VEL
LIN {X 0,Y 415.258,Z 240.873,A -85,B 0,C 180,E1 -10513.342,E2 -10513.342} C_VEL
LIN {X 0,Y 414.804,Z 250.23,A -85,B 0,C 180,E1 -10513.829,E2 -10513.829} C_VEL
LIN {X 0,Y 414.083,Z 260.37,A -85,B 0,C 180,E1 -10514.495,E2 -10514.495} C_VEL
LIN {X 0,Y 413.492,Z 269.368,A -85,B 0,C 180,E1 -10515.229,E2 -10515.229} C_VEL
LIN {X 0,Y 412.874,Z 277.248,A -85,B 0,C 180,E1 -10515.994,E2 -10515.994} C_VEL
LIN {X 0,Y 412.355,Z 285.495,A -85,B 0,C 180,E1 -10516.949,E2 -10516.949} C_VEL
LIN {X 0,Y 411.79,Z 292.715,A -85,B 0,C 180,E1 -10517.932,E2 -10517.932} C_VEL
LIN {X 0,Y 411.295,Z 298.916,A -85,B 0,C 180,E1 -10518.917,E2 -10518.917} C_VEL
LIN {X 0,Y 410.795,Z 305.453,A -85,B 0,C 180,E1 -10520.149,E2 -10520.149} C_VEL
LIN {X 0,Y 410.528,Z 309.956,A -85,B 0,C 180,E1 -10521.137,E2 -10521.137} C_VEL
LIN {X 0,Y 410.185,Z 315.445,A -85,B 0,C 180,E1 -10522.617,E2 -10522.617} C_VEL
LIN {X 0,Y 410.015,Z 319.769,A -85,B 0,C 180,E1 -10524.097,E2 -10524.097} C_VEL
LIN {X 0,Y 410.017,Z 322.137,A -85,B 0,C 180,E1 -10525.084,E2 -10525.084} C_VEL
LIN {X 0,Y 409.932,Z 323.933,A -85,B 0,C 180,E1 -10526.068,E2 -10526.068} C_VEL
LIN {X 0,Y 409.967,Z 326.377,A -85,B 0,C 180,E1 -10528.035,E2 -10528.035} C_VEL
LIN {X 0,Y 409.937,Z 326.964,A -85,B 0,C 180,E1 -10529.018,E2 -10529.018} C_VEL
LIN {X 0,Y 409.937,Z 326.964,A -85,B 0,C 180,E1 -10530.982,E2 -10530.982} C_VEL
LIN {X 0,Y 409.967,Z 326.377,A -85,B 0,C 180,E1 -10531.965,E2 -10531.965} C_VEL
LIN {X 0,Y 409.932,Z 323.933,A -85,B 0,C 180,E1 -10533.932,E2 -10533.932} C_VEL
LIN {X 0,Y 410.014,Z 320.986,A -85,B 0,C 180,E1 -10535.41,E2 -10535.41} C_VEL
LIN {X 0,Y 410.164,Z 317,A -85,B 0,C 180,E1 -10536.889,E2 -10536.889} C_VEL
LIN {X 0,Y 410.413,Z 311.871,A -85,B 0,C 180,E1 -10538.369,E2 -10538.369} C_VEL
LIN {X 0,Y 410.728,Z 306.609,A -85,B 0,C 180,E1 -10539.604,E2 -10539.604} C_VEL
LIN {X 0,Y 411.135,Z 300.291,A -85,B 0,C 180,E1 -10540.838,E2 -10540.838} C_VEL
LIN {X 0,Y 411.661,Z 294.342,A -85,B 0,C 180,E1 -10541.822,E2 -10541.822} C_VEL
LIN {X 0,Y 412.185,Z 287.414,A -85,B 0,C 180,E1 -10542.806,E2 -10542.806} C_VEL
LIN {X 0,Y 412.808,Z 279.233,A -85,B 0,C 180,E1 -10543.789,E2 -10543.789} C_VEL
LIN {X 0,Y 413.401,Z 270.686,A -85,B 0,C 180,E1 -10544.651,E2 -10544.651} C_VEL
LIN {X 0,Y 413.985,Z 262.002,A -85,B 0,C 180,E1 -10545.382,E2 -10545.382} C_VEL
LIN {X 0,Y 414.658,Z 252.244,A -85,B 0,C 180,E1 -10546.05,E2 -10546.05} C_VEL
LIN {X 0,Y 415.208,Z 242.161,A -85,B 0,C 180,E1 -10546.597,E2 -10546.597} C_VEL
LIN {X 0,Y 415.697,Z 232.647,A -85,B 0,C 180,E1 -10546.988,E2 -10546.988} C_VEL
LIN {X 0,Y 416.046,Z 222.333,A -85,B 0,C 180,E1 -10547.289,E2 -10547.289} C_VEL
LIN {X 0,Y 416.738,Z 165.806,A -85,B 0,C 180,E1 -10548.293,E2 -10548.293} C_VEL
LIN {X 0,Y 416.889,Z 142.756,A -85,B 0,C 180,E1 -10548.696,E2 -10548.696} C_VEL
LIN {X 0,Y 412.115,Z 116.682,A -85,B 0,C 180,E1 -10549.403,E2 -10549.403} C_VEL
LIN {X 0,Y 412.104,Z 115.598,A -85,B 0,C 180,E1 -10549.553,E2 -10549.553} C_VEL
LIN {X 0,Y 413.062,Z 102.348,A -85,B 0,C 180,E1 -10553.037,E2 -10553.037} C_VEL
LIN {X 0,Y 413.736,Z 92.972,A -85,B 0,C 180,E1 -10555.449,E2 -10555.449} C_VEL
LIN {X 0,Y 412.505,Z 84.969,A -85,B 0,C 180,E1 -10557.631,E2 -10557.631} C_VEL
LIN {X 0,Y 411.237,Z 78.775,A -85,B 0,C 180,E1 -10559.482,E2 -10559.482} C_VEL
LIN {X 0,Y 411.209,Z 78.763,A -85,B 0,C 180,E1 -10563.155,E2 -10563.155} C_VEL
LIN {X 0,Y 411.198,Z 78.762,A -85,B 0,C 180,E1 -10566.553,E2 -10566.553} C_VEL
LIN {X 0,Y 411.213,Z 78.745,A -85,B 0,C 180,E1 -10569.727,E2 -10569.727} C_VEL
LIN {X 0,Y 411.175,Z 78.768,A -85,B 0,C 180,E1 -10573.133,E2 -10573.133} C_VEL
LIN {X 0,Y 411.169,Z 78.767,A -85,B 0,C 180,E1 -10575.881,E2 -10575.881} C_VEL
LIN {X 0,Y 411.165,Z 78.767,A -85,B 0,C 180,E1 -10578.771,E2 -10578.771} C_VEL
LIN {X 0,Y 411.193,Z 78.763,A -85,B 0,C 180,E1 -10582.026,E2 -10582.026} C_VEL
LIN {X 0,Y 411.207,Z 78.748,A -85,B 0,C 180,E1 -10585.666,E2 -10585.666} C_VEL
LIN {X 0,Y 411.19,Z 78.767,A -85,B 0,C 180,E1 -10589.152,E2 -10589.152} C_VEL
LIN {X 0,Y 411.26,Z 78.742,A -85,B 0,C 180,E1 -10592.522,E2 -10592.522} C_VEL
LIN {X 0,Y 411.228,Z 78.755,A -85,B 0,C 180,E1 -10595.784,E2 -10595.784} C_VEL
LIN {X 0,Y 411.197,Z 78.755,A -85,B 0,C 180,E1 -10598.965,E2 -10598.965} C_VEL
LIN {X 0,Y 411.253,Z 78.736,A -85,B 0,C 180,E1 -10602.084,E2 -10602.084} C_VEL
LIN {X 0,Y 411.261,Z 78.753,A -85,B 0,C 180,E1 -10605.147,E2 -10605.147} C_VEL
LIN {X 0,Y 411.284,Z 78.744,A -85,B 0,C 180,E1 -10608.167,E2 -10608.167} C_VEL
LIN {X 0,Y 411.482,Z 78.716,A -85,B 0,C 180,E1 -10612.146,E2 -10612.146} C_VEL
LIN {X 0,Y 411.489,Z 78.728,A -85,B 0,C 180,E1 -10614.118,E2 -10614.118} C_VEL
LIN {X 0,Y 411.511,Z 78.714,A -85,B 0,C 180,E1 -10618.042,E2 -10618.042} C_VEL
LIN {X 0,Y 411.64,Z 78.686,A -85,B 0,C 180,E1 -10619.999,E2 -10619.999} C_VEL
LIN {X 0,Y 411.457,Z 78.724,A -85,B 0,C 180,E1 -10622.937,E2 -10622.937} C_VEL
LIN {X 0,Y 411.46,Z 78.726,A -85,B 0,C 180,E1 -10626.866,E2 -10626.866} C_VEL
LIN {X 0,Y 411.295,Z 78.73,A -85,B 0,C 180,E1 -10629.838,E2 -10629.838} C_VEL
LIN {X 0,Y 411.312,Z 78.745,A -85,B 0,C 180,E1 -10633.109,E2 -10633.109} C_VEL
LIN {X 0,Y 411.256,Z 78.752,A -85,B 0,C 180,E1 -10636.888,E2 -10636.888} C_VEL
LIN {X 0,Y 411.229,Z 78.747,A -85,B 0,C 180,E1 -10639.986,E2 -10639.986} C_VEL
LIN {X 0,Y 411.201,Z 78.766,A -85,B 0,C 180,E1 -10643.147,E2 -10643.147} C_VEL
LIN {X 0,Y 411.236,Z 78.748,A -85,B 0,C 180,E1 -10646.38,E2 -10646.38} C_VEL
LIN {X 0,Y 411.198,Z 78.761,A -85,B 0,C 180,E1 -10649.712,E2 -10649.712} C_VEL
LIN {X 0,Y 411.204,Z 78.755,A -85,B 0,C 180,E1 -10653.155,E2 -10653.155} C_VEL
LIN {X 0,Y 411.193,Z 78.763,A -85,B 0,C 180,E1 -10656.553,E2 -10656.553} C_VEL
LIN {X 0,Y 411.223,Z 78.754,A -85,B 0,C 180,E1 -10659.73,E2 -10659.73} C_VEL
LIN {X 0,Y 411.174,Z 78.766,A -85,B 0,C 180,E1 -10663.133,E2 -10663.133} C_VEL
LIN {X 0,Y 411.164,Z 78.756,A -85,B 0,C 180,E1 -10665.881,E2 -10665.881} C_VEL
LIN {X 0,Y 411.159,Z 78.741,A -85,B 0,C 180,E1 -10668.771,E2 -10668.771} C_VEL
LIN {X 0,Y 411.207,Z 78.763,A -85,B 0,C 180,E1 -10671.83,E2 -10671.83} C_VEL
LIN {X 0,Y 411.208,Z 78.74,A -85,B 0,C 180,E1 -10675.121,E2 -10675.121} C_VEL
LIN {X 0,Y 411.162,Z 78.771,A -85,B 0,C 180,E1 -10678.003,E2 -10678.003} C_VEL
LIN {X 0,Y 411.214,Z 78.751,A -85,B 0,C 180,E1 -10681.41,E2 -10681.41} C_VEL
LIN {X 0,Y 411.234,Z 78.762,A -85,B 0,C 180,E1 -10683.619,E2 -10683.619} C_VEL
LIN {X 0,Y 411.2,Z 78.765,A -85,B 0,C 180,E1 -10686.852,E2 -10686.852} C_VEL
LIN {X 0,Y 411.212,Z 78.765,A -85,B 0,C 180,E1 -10690.05,E2 -10690.05} C_VEL
LIN {X 0,Y 411.259,Z 78.76,A -85,B 0,C 180,E1 -10693.131,E2 -10693.131} C_VEL
LIN {X 0,Y 411.302,Z 78.754,A -85,B 0,C 180,E1 -10696.896,E2 -10696.896} C_VEL
LIN {X 0,Y 411.29,Z 78.755,A -85,B 0,C 180,E1 -10700.161,E2 -10700.161} C_VEL
LIN {X 0,Y 411.458,Z 78.735,A -85,B 0,C 180,E1 -10703.133,E2 -10703.133} C_VEL
LIN {X 0,Y 411.309,Z 78.753,A -85,B 0,C 180,E1 -10705.099,E2 -10705.099} C_VEL
LIN {X 0,Y 411.511,Z 78.727,A -85,B 0,C 180,E1 -10708.043,E2 -10708.043} C_VEL
LIN {X 0,Y 411.639,Z 78.712,A -85,B 0,C 180,E1 -10710,E2 -10710} C_VEL
LIN {X 0,Y 411.462,Z 78.734,A -85,B 0,C 180,E1 -10712.937,E2 -10712.937} C_VEL
LIN {X 0,Y 411.458,Z 78.735,A -85,B 0,C 180,E1 -10716.867,E2 -10716.867} C_VEL
LIN {X 0,Y 411.29,Z 78.755,A -85,B 0,C 180,E1 -10719.839,E2 -10719.839} C_VEL
LIN {X 0,Y 411.281,Z 78.755,A -85,B 0,C 180,E1 -10723.316,E2 -10723.316} C_VEL
LIN {X 0,Y 411.254,Z 78.76,A -85,B 0,C 180,E1 -10726.889,E2 -10726.889} C_VEL
LIN {X 0,Y 411.236,Z 78.76,A -85,B 0,C 180,E1 -10727.582,E2 -10727.582} C_VEL
LIN {X 0,Y 410.576,Z 78.845,A -85,B 0,C 180,E1 -10728.399,E2 -10728.399} C_VEL
LIN {X 0,Y 407.689,Z 79.204,A -85,B 0,C 180,E1 -10729.728,E2 -10729.728} C_VEL
LIN {X 0,Y 405.245,Z 79.508,A -85,B 0,C 180,E1 -10730.8,E2 -10730.8} C_VEL
LIN {X 0,Y 404.209,Z 79.637,A -85,B 0,C 180,E1 -10731.631,E2 -10731.631} C_VEL
LIN {X 0,Y 404.132,Z 79.644,A -85,B 0,C 180,E1 -10731.912,E2 -10731.912} C_VEL
LIN {X 0,Y 404.212,Z 79.634,A -85,B 0,C 180,E1 -10735.297,E2 -10735.297} C_VEL
LIN {X 0,Y 404.192,Z 79.632,A -85,B 0,C 180,E1 -10738,E2 -10738} C_VEL
LIN {X 0,Y 404.138,Z 79.644,A -85,B 0,C 180,E1 -10741.559,E2 -10741.559} C_VEL
LIN {X 0,Y 404.182,Z 79.612,A -85,B 0,C 180,E1 -10745.016,E2 -10745.016} C_VEL
LIN {X 0,Y 404.154,Z 79.64,A -85,B 0,C 180,E1 -10748.757,E2 -10748.757} C_VEL
LIN {X 0,Y 404.119,Z 79.613,A -85,B 0,C 180,E1 -10751.6,E2 -10751.6} C_VEL
LIN {X 0,Y 404.141,Z 79.633,A -85,B 0,C 180,E1 -10754.522,E2 -10754.522} C_VEL
LIN {X 0,Y 404.167,Z 79.642,A -85,B 0,C 180,E1 -10757.3,E2 -10757.3} C_VEL
LIN {X 0,Y 404.166,Z 79.634,A -85,B 0,C 180,E1 -10759.956,E2 -10759.956} C_VEL
LIN {X 0,Y 404.138,Z 79.646,A -85,B 0,C 180,E1 -10763.125,E2 -10763.125} C_VEL
LIN {X 0,Y 404.142,Z 79.631,A -85,B 0,C 180,E1 -10766.188,E2 -10766.188} C_VEL
LIN {X 0,Y 404.143,Z 79.64,A -85,B 0,C 180,E1 -10769.715,E2 -10769.715} C_VEL
LIN {X 0,Y 404.193,Z 79.622,A -85,B 0,C 180,E1 -10773.123,E2 -10773.123} C_VEL
LIN {X 0,Y 404.175,Z 79.638,A -85,B 0,C 180,E1 -10775.335,E2 -10775.335} C_VEL
LIN {X 0,Y 404.158,Z 79.637,A -85,B 0,C 180,E1 -10778.582,E2 -10778.582} C_VEL
LIN {X 0,Y 404.209,Z 79.615,A -85,B 0,C 180,E1 -10781.762,E2 -10781.762} C_VEL
LIN {X 0,Y 404.207,Z 79.636,A -85,B 0,C 180,E1 -10784.883,E2 -10784.883} C_VEL
LIN {X 0,Y 404.268,Z 79.622,A -85,B 0,C 180,E1 -10787.959,E2 -10787.959} C_VEL
LIN {X 0,Y 404.433,Z 79.594,A -85,B 0,C 180,E1 -10792.1,E2 -10792.1} C_VEL
LIN {X 0,Y 404.423,Z 79.606,A -85,B 0,C 180,E1 -10794.016,E2 -10794.016} C_VEL
LIN {X 0,Y 404.48,Z 79.588,A -85,B 0,C 180,E1 -10798.009,E2 -10798.009} C_VEL
LIN {X 0,Y 404.609,Z 79.561,A -85,B 0,C 180,E1 -10800.001,E2 -10800.001} C_VEL
LIN {X 0,Y 404.415,Z 79.602,A -85,B 0,C 180,E1 -10802.989,E2 -10802.989} C_VEL
LIN {X 0,Y 404.435,Z 79.605,A -85,B 0,C 180,E1 -10805.985,E2 -10805.985} C_VEL
LIN {X 0,Y 404.423,Z 79.593,A -85,B 0,C 180,E1 -10807.992,E2 -10807.992} C_VEL
LIN {X 0,Y 404.256,Z 79.623,A -85,B 0,C 180,E1 -10812.042,E2 -10812.042} C_VEL
LIN {X 0,Y 404.207,Z 79.633,A -85,B 0,C 180,E1 -10815.118,E2 -10815.118} C_VEL
LIN {X 0,Y 404.211,Z 79.611,A -85,B 0,C 180,E1 -10818.239,E2 -10818.239} C_VEL
LIN {X 0,Y 404.161,Z 79.636,A -85,B 0,C 180,E1 -10821.419,E2 -10821.419} C_VEL
LIN {X 0,Y 404.178,Z 79.635,A -85,B 0,C 180,E1 -10824.666,E2 -10824.666} C_VEL
LIN {X 0,Y 404.196,Z 79.624,A -85,B 0,C 180,E1 -10828,E2 -10828} C_VEL
LIN {X 0,Y 404.14,Z 79.641,A -85,B 0,C 180,E1 -10831.558,E2 -10831.558} C_VEL
LIN {X 0,Y 404.186,Z 79.627,A -85,B 0,C 180,E1 -10835.017,E2 -10835.017} C_VEL
LIN {X 0,Y 404.152,Z 79.639,A -85,B 0,C 180,E1 -10838.758,E2 -10838.758} C_VEL
LIN {X 0,Y 404.124,Z 79.642,A -85,B 0,C 180,E1 -10841.6,E2 -10841.6} C_VEL
LIN {X 0,Y 404.147,Z 79.638,A -85,B 0,C 180,E1 -10844.522,E2 -10844.522} C_VEL
LIN {X 0,Y 404.138,Z 79.641,A -85,B 0,C 180,E1 -10847.296,E2 -10847.296} C_VEL
LIN {X 0,Y 404.171,Z 79.62,A -85,B 0,C 180,E1 -10849.956,E2 -10849.956} C_VEL
LIN {X 0,Y 404.142,Z 79.641,A -85,B 0,C 180,E1 -10853.125,E2 -10853.125} C_VEL
LIN {X 0,Y 404.148,Z 79.644,A -85,B 0,C 180,E1 -10856.188,E2 -10856.188} C_VEL
LIN {X 0,Y 404.194,Z 79.633,A -85,B 0,C 180,E1 -10860.101,E2 -10860.101} C_VEL
LIN {X 0,Y 404.257,Z 79.904,A -85,B 0,C 180,E1 -10860.372,E2 -10860.372} C_VEL
LIN {X 0,Y 406.11,Z 89.516,A -85,B 0,C 180,E1 -10863.26,E2 -10863.26} C_VEL
LIN {X 0,Y 406.729,Z 94.728,A -85,B 0,C 180,E1 -10864.681,E2 -10864.681} C_VEL
LIN {X 0,Y 405.762,Z 108.144,A -85,B 0,C 180,E1 -10868.137,E2 -10868.137} C_VEL
LIN {X 0,Y 405.142,Z 115.97,A -85,B 0,C 180,E1 -10870.202,E2 -10870.202} C_VEL
LIN {X 0,Y 405.927,Z 120.282,A -85,B 0,C 180,E1 -10870.373,E2 -10870.373} C_VEL
LIN {X 0,Y 410.175,Z 144.065,A -85,B 0,C 180,E1 -10871.014,E2 -10871.014} C_VEL
LIN {X 0,Y 409.344,Z 220.812,A -85,B 0,C 180,E1 -10872.386,E2 -10872.386} C_VEL
LIN {X 0,Y 408.964,Z 231.583,A -85,B 0,C 180,E1 -10872.692,E2 -10872.692} C_VEL
LIN {X 0,Y 408.468,Z 240.682,A -85,B 0,C 180,E1 -10873.057,E2 -10873.057} C_VEL
LIN {X 0,Y 407.982,Z 250.04,A -85,B 0,C 180,E1 -10873.551,E2 -10873.551} C_VEL
LIN {X 0,Y 407.225,Z 260.179,A -85,B 0,C 180,E1 -10874.228,E2 -10874.228} C_VEL
LIN {X 0,Y 406.606,Z 269.177,A -85,B 0,C 180,E1 -10874.973,E2 -10874.973} C_VEL
LIN {X 0,Y 405.878,Z 278.005,A -85,B 0,C 180,E1 -10875.854,E2 -10875.854} C_VEL
LIN {X 0,Y 405.381,Z 285.357,A -85,B 0,C 180,E1 -10876.727,E2 -10876.727} C_VEL
LIN {X 0,Y 404.803,Z 292.523,A -85,B 0,C 180,E1 -10877.721,E2 -10877.721} C_VEL
LIN {X 0,Y 404.299,Z 298.725,A -85,B 0,C 180,E1 -10878.723,E2 -10878.723} C_VEL
LIN {X 0,Y 403.767,Z 305.262,A -85,B 0,C 180,E1 -10879.976,E2 -10879.976} C_VEL
LIN {X 0,Y 403.484,Z 309.764,A -85,B 0,C 180,E1 -10880.981,E2 -10880.981} C_VEL
LIN {X 0,Y 403.132,Z 315.255,A -85,B 0,C 180,E1 -10882.487,E2 -10882.487} C_VEL
LIN {X 0,Y 402.94,Z 319.578,A -85,B 0,C 180,E1 -10883.993,E2 -10883.993} C_VEL
LIN {X 0,Y 402.929,Z 321.946,A -85,B 0,C 180,E1 -10884.997,E2 -10884.997} C_VEL
LIN {X 0,Y 402.852,Z 323.742,A -85,B 0,C 180,E1 -10885.999,E2 -10885.999} C_VEL
LIN {X 0,Y 402.865,Z 326.186,A -85,B 0,C 180,E1 -10888.001,E2 -10888.001} C_VEL
LIN {X 0,Y 402.864,Z 326.775,A -85,B 0,C 180,E1 -10889,E2 -10889} C_VEL
LIN {X 0,Y 402.864,Z 326.775,A -85,B 0,C 180,E1 -10891,E2 -10891} C_VEL
LIN {X 0,Y 402.865,Z 326.186,A -85,B 0,C 180,E1 -10891.999,E2 -10891.999} C_VEL
LIN {X 0,Y 402.852,Z 323.742,A -85,B 0,C 180,E1 -10894.001,E2 -10894.001} C_VEL
LIN {X 0,Y 402.912,Z 320.795,A -85,B 0,C 180,E1 -10895.505,E2 -10895.505} C_VEL
LIN {X 0,Y 403.076,Z 316.809,A -85,B 0,C 180,E1 -10897.01,E2 -10897.01} C_VEL
LIN {X 0,Y 403.355,Z 311.68,A -85,B 0,C 180,E1 -10898.517,E2 -10898.517} C_VEL
LIN {X 0,Y 403.69,Z 306.418,A -85,B 0,C 180,E1 -10899.773,E2 -10899.773} C_VEL
LIN {X 0,Y 404.135,Z 300.1,A -85,B 0,C 180,E1 -10901.028,E2 -10901.028} C_VEL
LIN {X 0,Y 404.668,Z 294.15,A -85,B 0,C 180,E1 -10902.029,E2 -10902.029} C_VEL
LIN {X 0,Y 405.232,Z 287.222,A -85,B 0,C 180,E1 -10903.03,E2 -10903.03} C_VEL
LIN {X 0,Y 405.865,Z 279.042,A -85,B 0,C 180,E1 -10904.03,E2 -10904.03} C_VEL
LIN {X 0,Y 406.49,Z 270.664,A -85,B 0,C 180,E1 -10904.89,E2 -10904.89} C_VEL
LIN {X 0,Y 407.124,Z 261.811,A -85,B 0,C 180,E1 -10905.648,E2 -10905.648} C_VEL
LIN {X 0,Y 407.842,Z 252.054,A -85,B 0,C 180,E1 -10906.326,E2 -10906.326} C_VEL
LIN {X 0,Y 408.408,Z 241.97,A -85,B 0,C 180,E1 -10906.881,E2 -10906.881} C_VEL
LIN {X 0,Y 408.924,Z 232.457,A -85,B 0,C 180,E1 -10907.278,E2 -10907.278} C_VEL
LIN {X 0,Y 409.285,Z 222.143,A -85,B 0,C 180,E1 -10907.584,E2 -10907.584} C_VEL
LIN {X 0,Y 410.009,Z 165.616,A -85,B 0,C 180,E1 -10908.604,E2 -10908.604} C_VEL
LIN {X 0,Y 410.096,Z 143.366,A -85,B 0,C 180,E1 -10909.003,E2 -10909.003} C_VEL
LIN {X 0,Y 405.187,Z 116.42,A -85,B 0,C 180,E1 -10909.753,E2 -10909.753} C_VEL
LIN {X 0,Y 405.196,Z 115.41,A -85,B 0,C 180,E1 -10909.901,E2 -10909.901} C_VEL
LIN {X 0,Y 406.384,Z 100.175,A -85,B 0,C 180,E1 -10913.979,E2 -10913.979} C_VEL
LIN {X 0,Y 406.767,Z 94.026,A -85,B 0,C 180,E1 -10915.591,E2 -10915.591} C_VEL
LIN {X 0,Y 405.436,Z 85.759,A -85,B 0,C 180,E1 -10917.906,E2 -10917.906} C_VEL
LIN {X 0,Y 404.228,Z 79.65,A -85,B 0,C 180,E1 -10919.752,E2 -10919.752} C_VEL
LIN {X 0,Y 404.173,Z 79.641,A -85,B 0,C 180,E1 -10923.42,E2 -10923.42} C_VEL
LIN {X 0,Y 404.146,Z 79.638,A -85,B 0,C 180,E1 -10926.246,E2 -10926.246} C_VEL
LIN {X 0,Y 404.157,Z 79.636,A -85,B 0,C 180,E1 -10928.757,E2 -10928.757} C_VEL
LIN {X 0,Y 404.124,Z 79.636,A -85,B 0,C 180,E1 -10931.599,E2 -10931.599} C_VEL
LIN {X 0,Y 404.147,Z 79.638,A -85,B 0,C 180,E1 -10934.522,E2 -10934.522} C_VEL
LIN {X 0,Y 404.138,Z 79.647,A -85,B 0,C 180,E1 -10937.295,E2 -10937.295} C_VEL
LIN {X 0,Y 404.17,Z 79.63,A -85,B 0,C 180,E1 -10939.955,E2 -10939.955} C_VEL
LIN {X 0,Y 404.137,Z 79.646,A -85,B 0,C 180,E1 -10943.125,E2 -10943.125} C_VEL
LIN {X 0,Y 404.146,Z 79.627,A -85,B 0,C 180,E1 -10946.187,E2 -10946.187} C_VEL
LIN {X 0,Y 404.147,Z 79.64,A -85,B 0,C 180,E1 -10949.714,E2 -10949.714} C_VEL
LIN {X 0,Y 404.196,Z 79.62,A -85,B 0,C 180,E1 -10953.122,E2 -10953.122} C_VEL
LIN {X 0,Y 404.178,Z 79.635,A -85,B 0,C 180,E1 -10955.334,E2 -10955.334} C_VEL
LIN {X 0,Y 404.161,Z 79.636,A -85,B 0,C 180,E1 -10958.581,E2 -10958.581} C_VEL
LIN {X 0,Y 404.211,Z 79.611,A -85,B 0,C 180,E1 -10961.761,E2 -10961.761} C_VEL
LIN {X 0,Y 404.207,Z 79.633,A -85,B 0,C 180,E1 -10964.882,E2 -10964.882} C_VEL
LIN {X 0,Y 404.256,Z 79.623,A -85,B 0,C 180,E1 -10967.958,E2 -10967.958} C_VEL
LIN {X 0,Y 404.434,Z 79.592,A -85,B 0,C 180,E1 -10972.099,E2 -10972.099} C_VEL
LIN {X 0,Y 404.435,Z 79.605,A -85,B 0,C 180,E1 -10974.015,E2 -10974.015} C_VEL
LIN {X 0,Y 404.48,Z 79.589,A -85,B 0,C 180,E1 -10978.008,E2 -10978.008} C_VEL
LIN {X 0,Y 404.609,Z 79.561,A -85,B 0,C 180,E1 -10979.999,E2 -10979.999} C_VEL
LIN {X 0,Y 404.415,Z 79.601,A -85,B 0,C 180,E1 -10982.988,E2 -10982.988} C_VEL
LIN {X 0,Y 404.411,Z 79.604,A -85,B 0,C 180,E1 -10986.987,E2 -10986.987} C_VEL
LIN {X 0,Y 404.261,Z 79.606,A -85,B 0,C 180,E1 -10990.011,E2 -10990.011} C_VEL
LIN {X 0,Y 404.265,Z 79.624,A -85,B 0,C 180,E1 -10993.211,E2 -10993.211} C_VEL
LIN {X 0,Y 404.214,Z 79.629,A -85,B 0,C 180,E1 -10997.007,E2 -10997.007} C_VEL
LIN {X 0,Y 404.162,Z 79.627,A -85,B 0,C 180,E1 -11000.351,E2 -11000.351} C_VEL
LIN {X 0,Y 404.167,Z 79.639,A -85,B 0,C 180,E1 -11003.574,E2 -11003.574} C_VEL
LIN {X 0,Y 404.181,Z 79.627,A -85,B 0,C 180,E1 -11005.766,E2 -11005.766} C_VEL
LIN {X 0,Y 404.193,Z 79.622,A -85,B 0,C 180,E1 -11007.999,E2 -11007.999} C_VEL
LIN {X 0,Y 404.137,Z 79.642,A -85,B 0,C 180,E1 -11011.558,E2 -11011.558} C_VEL
LIN {X 0,Y 404.183,Z 79.628,A -85,B 0,C 180,E1 -11015.016,E2 -11015.016} C_VEL
LIN {X 0,Y 404.159,Z 79.64,A -85,B 0,C 180,E1 -11018.756,E2 -11018.756} C_VEL
LIN {X 0,Y 404.146,Z 79.635,A -85,B 0,C 180,E1 -11021.604,E2 -11021.604} C_VEL
LIN {X 0,Y 404.142,Z 79.64,A -85,B 0,C 180,E1 -11024.522,E2 -11024.522} C_VEL
LIN {X 0,Y 404.132,Z 79.613,A -85,B 0,C 180,E1 -11027.295,E2 -11027.295} C_VEL
LIN {X 0,Y 404.165,Z 79.626,A -85,B 0,C 180,E1 -11029.955,E2 -11029.955} C_VEL
LIN {X 0,Y 404.136,Z 79.64,A -85,B 0,C 180,E1 -11033.124,E2 -11033.124} C_VEL
LIN {X 0,Y 404.141,Z 79.625,A -85,B 0,C 180,E1 -11036.188,E2 -11036.188} C_VEL
LIN {X 0,Y 404.142,Z 79.634,A -85,B 0,C 180,E1 -11039.715,E2 -11039.715} C_VEL
LIN {X 0,Y 404.192,Z 79.637,A -85,B 0,C 180,E1 -11043.123,E2 -11043.123} C_VEL
LIN {X 0,Y 404.174,Z 79.641,A -85,B 0,C 180,E1 -11045.334,E2 -11045.334} C_VEL
LIN {X 0,Y 404.135,Z 79.645,A -85,B 0,C 180,E1 -11048.581,E2 -11048.581} C_VEL
LIN {X 0,Y 404.207,Z 79.638,A -85,B 0,C 180,E1 -11051.762,E2 -11051.762} C_VEL
LIN {X 0,Y 404.203,Z 79.637,A -85,B 0,C 180,E1 -11054.882,E2 -11054.882} C_VEL
LIN {X 0,Y 404.253,Z 79.632,A -85,B 0,C 180,E1 -11057.958,E2 -11057.958} C_VEL
LIN {X 0,Y 404.43,Z 79.61,A -85,B 0,C 180,E1 -11062.1,E2 -11062.1} C_VEL
LIN {X 0,Y 404.422,Z 79.61,A -85,B 0,C 180,E1 -11064.015,E2 -11064.015} C_VEL
LIN {X 0,Y 404.479,Z 79.603,A -85,B 0,C 180,E1 -11068.009,E2 -11068.009} C_VEL
LIN {X 0,Y 404.608,Z 79.588,A -85,B 0,C 180,E1 -11070,E2 -11070} C_VEL
LIN {X 0,Y 404.42,Z 79.611,A -85,B 0,C 180,E1 -11072.988,E2 -11072.988} C_VEL
LIN {X 0,Y 404.409,Z 79.613,A -85,B 0,C 180,E1 -11076.987,E2 -11076.987} C_VEL
LIN {X 0,Y 404.255,Z 79.631,A -85,B 0,C 180,E1 -11080.012,E2 -11080.012} C_VEL
LIN {X 0,Y 404.263,Z 79.631,A -85,B 0,C 180,E1 -11083.211,E2 -11083.211} C_VEL
LIN {X 0,Y 404.212,Z 79.636,A -85,B 0,C 180,E1 -11087.007,E2 -11087.007} C_VEL
LIN {X 0,Y 404.16,Z 79.644,A -85,B 0,C 180,E1 -11090.352,E2 -11090.352} C_VEL
LIN {X 0,Y 404.132,Z 79.644,A -85,B 0,C 180,E1 -11091.912,E2 -11091.912} C_VEL
LIN {X 0,Y 403.49,Z 79.728,A -85,B 0,C 180,E1 -11092.743,E2 -11092.743} C_VEL
LIN {X 0,Y 400.658,Z 80.085,A -85,B 0,C 180,E1 -11094.095,E2 -11094.095} C_VEL
LIN {X 0,Y 398.249,Z 80.386,A -85,B 0,C 180,E1 -11095.187,E2 -11095.187} C_VEL
LIN {X 0,Y 397.214,Z 80.511,A -85,B 0,C 180,E1 -11096.031,E2 -11096.031} C_VEL
LIN {X 0,Y 397.131,Z 80.519,A -85,B 0,C 180,E1 -11096.317,E2 -11096.317} C_VEL
LIN {X 0,Y 397.118,Z 80.506,A -85,B 0,C 180,E1 -11098.544,E2 -11098.544} C_VEL
LIN {X 0,Y 397.077,Z 80.524,A -85,B 0,C 180,E1 -11102.072,E2 -11102.072} C_VEL
LIN {X 0,Y 397.116,Z 80.495,A -85,B 0,C 180,E1 -11105.504,E2 -11105.504} C_VEL
LIN {X 0,Y 397.129,Z 80.515,A -85,B 0,C 180,E1 -11108.862,E2 -11108.862} C_VEL
LIN {X 0,Y 397.064,Z 80.489,A -85,B 0,C 180,E1 -11112.268,E2 -11112.268} C_VEL
LIN {X 0,Y 397.083,Z 80.514,A -85,B 0,C 180,E1 -11115.069,E2 -11115.069} C_VEL
LIN {X 0,Y 397.106,Z 80.513,A -85,B 0,C 180,E1 -11118.015,E2 -11118.015} C_VEL
LIN {X 0,Y 397.133,Z 80.514,A -85,B 0,C 180,E1 -11121.138,E2 -11121.138} C_VEL
LIN {X 0,Y 397.117,Z 80.512,A -85,B 0,C 180,E1 -11124.497,E2 -11124.497} C_VEL
LIN {X 0,Y 397.075,Z 80.521,A -85,B 0,C 180,E1 -11127.929,E2 -11127.929} C_VEL
LIN {X 0,Y 397.119,Z 80.505,A -85,B 0,C 180,E1 -11131.457,E2 -11131.457} C_VEL
LIN {X 0,Y 397.151,Z 80.504,A -85,B 0,C 180,E1 -11134.488,E2 -11134.488} C_VEL
LIN {X 0,Y 397.107,Z 80.517,A -85,B 0,C 180,E1 -11138.183,E2 -11138.183} C_VEL
LIN {X 0,Y 397.161,Z 80.493,A -85,B 0,C 180,E1 -11141.427,E2 -11141.427} C_VEL
LIN {X 0,Y 397.179,Z 80.512,A -85,B 0,C 180,E1 -11144.609,E2 -11144.609} C_VEL
LIN {X 0,Y 397.228,Z 80.498,A -85,B 0,C 180,E1 -11147.743,E2 -11147.743} C_VEL
LIN {X 0,Y 397.394,Z 80.469,A -85,B 0,C 180,E1 -11152.041,E2 -11152.041} C_VEL
LIN {X 0,Y 397.254,Z 80.499,A -85,B 0,C 180,E1 -11154.926,E2 -11154.926} C_VEL
LIN {X 0,Y 397.449,Z 80.464,A -85,B 0,C 180,E1 -11157.974,E2 -11157.974} C_VEL
LIN {X 0,Y 397.578,Z 80.436,A -85,B 0,C 180,E1 -11160.001,E2 -11160.001} C_VEL
LIN {X 0,Y 397.375,Z 80.479,A -85,B 0,C 180,E1 -11163.042,E2 -11163.042} C_VEL
LIN {X 0,Y 397.385,Z 80.482,A -85,B 0,C 180,E1 -11166.092,E2 -11166.092} C_VEL
LIN {X 0,Y 397.377,Z 80.468,A -85,B 0,C 180,E1 -11168.134,E2 -11168.134} C_VEL
LIN {X 0,Y 397.22,Z 80.498,A -85,B 0,C 180,E1 -11172.259,E2 -11172.259} C_VEL
LIN {X 0,Y 397.18,Z 80.51,A -85,B 0,C 180,E1 -11175.393,E2 -11175.393} C_VEL
LIN {X 0,Y 397.163,Z 80.488,A -85,B 0,C 180,E1 -11178.574,E2 -11178.574} C_VEL
LIN {X 0,Y 397.11,Z 80.516,A -85,B 0,C 180,E1 -11181.818,E2 -11181.818} C_VEL
LIN {X 0,Y 397.154,Z 80.501,A -85,B 0,C 180,E1 -11185.513,E2 -11185.513} C_VEL
LIN {X 0,Y 397.123,Z 80.506,A -85,B 0,C 180,E1 -11188.544,E2 -11188.544} C_VEL
LIN {X 0,Y 397.079,Z 80.519,A -85,B 0,C 180,E1 -11192.072,E2 -11192.072} C_VEL
LIN {X 0,Y 397.121,Z 80.513,A -85,B 0,C 180,E1 -11195.504,E2 -11195.504} C_VEL
LIN {X 0,Y 397.128,Z 80.512,A -85,B 0,C 180,E1 -11198.861,E2 -11198.861} C_VEL
LIN {X 0,Y 397.07,Z 80.524,A -85,B 0,C 180,E1 -11202.268,E2 -11202.268} C_VEL
LIN {X 0,Y 397.089,Z 80.517,A -85,B 0,C 180,E1 -11205.069,E2 -11205.069} C_VEL
LIN {X 0,Y 397.068,Z 80.521,A -85,B 0,C 180,E1 -11208.022,E2 -11208.022} C_VEL
LIN {X 0,Y 397.132,Z 80.508,A -85,B 0,C 180,E1 -11211.139,E2 -11211.139} C_VEL
LIN {X 0,Y 397.122,Z 80.506,A -85,B 0,C 180,E1 -11214.497,E2 -11214.497} C_VEL
LIN {X 0,Y 397.081,Z 80.515,A -85,B 0,C 180,E1 -11217.929,E2 -11217.929} C_VEL
LIN {X 0,Y 397.164,Z 80.636,A -85,B 0,C 180,E1 -11220.02,E2 -11220.02} C_VEL
LIN {X 0,Y 399.059,Z 90.384,A -85,B 0,C 180,E1 -11223.032,E2 -11223.032} C_VEL
LIN {X 0,Y 399.775,Z 95.598,A -85,B 0,C 180,E1 -11224.488,E2 -11224.488} C_VEL
LIN {X 0,Y 398.893,Z 106.98,A -85,B 0,C 180,E1 -11227.468,E2 -11227.468} C_VEL
LIN {X 0,Y 398.219,Z 115.765,A -85,B 0,C 180,E1 -11229.84,E2 -11229.84} C_VEL
LIN {X 0,Y 398.881,Z 119.62,A -85,B 0,C 180,E1 -11230.003,E2 -11230.003} C_VEL
LIN {X 0,Y 403.498,Z 145.116,A -85,B 0,C 180,E1 -11230.71,E2 -11230.71} C_VEL
LIN {X 0,Y 402.593,Z 220.622,A -85,B 0,C 180,E1 -11232.081,E2 -11232.081} C_VEL
LIN {X 0,Y 402.192,Z 231.392,A -85,B 0,C 180,E1 -11232.391,E2 -11232.391} C_VEL
LIN {X 0,Y 401.689,Z 240.492,A -85,B 0,C 180,E1 -11232.762,E2 -11232.762} C_VEL
LIN {X 0,Y 401.116,Z 250.856,A -85,B 0,C 180,E1 -11233.327,E2 -11233.327} C_VEL
LIN {X 0,Y 400.394,Z 259.988,A -85,B 0,C 180,E1 -11233.951,E2 -11233.951} C_VEL
LIN {X 0,Y 399.729,Z 268.986,A -85,B 0,C 180,E1 -11234.709,E2 -11234.709} C_VEL
LIN {X 0,Y 398.978,Z 277.829,A -85,B 0,C 180,E1 -11235.606,E2 -11235.606} C_VEL
LIN {X 0,Y 398.411,Z 285.343,A -85,B 0,C 180,E1 -11236.515,E2 -11236.515} C_VEL
LIN {X 0,Y 397.839,Z 292.332,A -85,B 0,C 180,E1 -11237.502,E2 -11237.502} C_VEL
LIN {X 0,Y 397.282,Z 298.533,A -85,B 0,C 180,E1 -11238.521,E2 -11238.521} C_VEL
LIN {X 0,Y 396.752,Z 305.07,A -85,B 0,C 180,E1 -11239.797,E2 -11239.797} C_VEL
LIN {X 0,Y 396.414,Z 309.572,A -85,B 0,C 180,E1 -11240.819,E2 -11240.819} C_VEL
LIN {X 0,Y 396.062,Z 315.063,A -85,B 0,C 180,E1 -11242.352,E2 -11242.352} C_VEL
LIN {X 0,Y 395.863,Z 319.387,A -85,B 0,C 180,E1 -11243.885,E2 -11243.885} C_VEL
LIN {X 0,Y 395.842,Z 321.755,A -85,B 0,C 180,E1 -11244.907,E2 -11244.907} C_VEL
LIN {X 0,Y 395.775,Z 323.552,A -85,B 0,C 180,E1 -11245.927,E2 -11245.927} C_VEL
LIN {X 0,Y 395.763,Z 325.996,A -85,B 0,C 180,E1 -11247.965,E2 -11247.965} C_VEL
LIN {X 0,Y 395.793,Z 326.585,A -85,B 0,C 180,E1 -11248.983,E2 -11248.983} C_VEL
LIN {X 0,Y 395.793,Z 326.585,A -85,B 0,C 180,E1 -11251.017,E2 -11251.017} C_VEL
LIN {X 0,Y 395.763,Z 325.996,A -85,B 0,C 180,E1 -11252.035,E2 -11252.035} C_VEL
LIN {X 0,Y 395.775,Z 323.552,A -85,B 0,C 180,E1 -11254.073,E2 -11254.073} C_VEL
LIN {X 0,Y 395.842,Z 321.755,A -85,B 0,C 180,E1 -11255.093,E2 -11255.093} C_VEL
LIN {X 0,Y 395.92,Z 318.149,A -85,B 0,C 180,E1 -11256.625,E2 -11256.625} C_VEL
LIN {X 0,Y 396.178,Z 313.404,A -85,B 0,C 180,E1 -11258.159,E2 -11258.159} C_VEL
LIN {X 0,Y 396.592,Z 307.382,A -85,B 0,C 180,E1 -11259.692,E2 -11259.692} C_VEL
LIN {X 0,Y 397.02,Z 301.284,A -85,B 0,C 180,E1 -11260.97,E2 -11260.97} C_VEL
LIN {X 0,Y 397.572,Z 295.586,A -85,B 0,C 180,E1 -11261.988,E2 -11261.988} C_VEL
LIN {X 0,Y 398.278,Z 287.031,A -85,B 0,C 180,E1 -11263.262,E2 -11263.262} C_VEL
LIN {X 0,Y 398.955,Z 278.85,A -85,B 0,C 180,E1 -11264.278,E2 -11264.278} C_VEL
LIN {X 0,Y 399.604,Z 270.472,A -85,B 0,C 180,E1 -11265.153,E2 -11265.153} C_VEL
LIN {X 0,Y 400.281,Z 261.62,A -85,B 0,C 180,E1 -11265.923,E2 -11265.923} C_VEL
LIN {X 0,Y 401.014,Z 251.862,A -85,B 0,C 180,E1 -11266.612,E2 -11266.612} C_VEL
LIN {X 0,Y 401.635,Z 241.78,A -85,B 0,C 180,E1 -11267.175,E2 -11267.175} C_VEL
LIN {X 0,Y 402.164,Z 232.267,A -85,B 0,C 180,E1 -11267.578,E2 -11267.578} C_VEL
LIN {X 0,Y 402.528,Z 221.953,A -85,B 0,C 180,E1 -11267.889,E2 -11267.889} C_VEL
LIN {X 0,Y 403.144,Z 175.468,A -85,B 0,C 180,E1 -11268.748,E2 -11268.748} C_VEL
LIN {X 0,Y 403.521,Z 145.11,A -85,B 0,C 180,E1 -11269.289,E2 -11269.289} C_VEL
LIN {X 0,Y 398.286,Z 116.246,A -85,B 0,C 180,E1 -11270.109,E2 -11270.109} C_VEL
LIN {X 0,Y 398.243,Z 115.223,A -85,B 0,C 180,E1 -11270.263,E2 -11270.263} C_VEL
LIN {X 0,Y 399.441,Z 100.993,A -85,B 0,C 180,E1 -11274.147,E2 -11274.147} C_VEL
LIN {X 0,Y 399.783,Z 94.886,A -85,B 0,C 180,E1 -11275.791,E2 -11275.791} C_VEL
LIN {X 0,Y 398.416,Z 86.773,A -85,B 0,C 180,E1 -11278.115,E2 -11278.115} C_VEL
LIN {X 0,Y 397.149,Z 80.534,A -85,B 0,C 180,E1 -11280.038,E2 -11280.038} C_VEL
LIN {X 0,Y 397.121,Z 80.521,A -85,B 0,C 180,E1 -11283.718,E2 -11283.718} C_VEL
LIN {X 0,Y 397.099,Z 80.52,A -85,B 0,C 180,E1 -11287.209,E2 -11287.209} C_VEL
LIN {X 0,Y 397.103,Z 80.5,A -85,B 0,C 180,E1 -11290.445,E2 -11290.445} C_VEL
LIN {X 0,Y 397.103,Z 80.521,A -85,B 0,C 180,E1 -11293.648,E2 -11293.648} C_VEL
LIN {X 0,Y 397.104,Z 80.518,A -85,B 0,C 180,E1 -11296.521,E2 -11296.521} C_VEL
LIN {X 0,Y 397.114,Z 80.508,A -85,B 0,C 180,E1 -11300.422,E2 -11300.422} C_VEL
LIN {X 0,Y 397.109,Z 80.513,A -85,B 0,C 180,E1 -11304.265,E2 -11304.265} C_VEL
LIN {X 0,Y 397.116,Z 80.506,A -85,B 0,C 180,E1 -11306.727,E2 -11306.727} C_VEL
LIN {X 0,Y 397.126,Z 80.515,A -85,B 0,C 180,E1 -11310.295,E2 -11310.295} C_VEL
LIN {X 0,Y 397.195,Z 80.492,A -85,B 0,C 180,E1 -11312.609,E2 -11312.609} C_VEL
LIN {X 0,Y 397.134,Z 80.511,A -85,B 0,C 180,E1 -11315.981,E2 -11315.981} C_VEL
LIN {X 0,Y 397.139,Z 80.502,A -85,B 0,C 180,E1 -11319.704,E2 -11319.704} C_VEL
LIN {X 0,Y 397.182,Z 80.498,A -85,B 0,C 180,E1 -11322.844,E2 -11322.844} C_VEL
LIN {X 0,Y 397.229,Z 80.5,A -85,B 0,C 180,E1 -11326.702,E2 -11326.702} C_VEL
LIN {X 0,Y 397.218,Z 80.483,A -85,B 0,C 180,E1 -11329.808,E2 -11329.808} C_VEL
LIN {X 0,Y 397.364,Z 80.481,A -85,B 0,C 180,E1 -11332.888,E2 -11332.888} C_VEL
LIN {X 0,Y 397.257,Z 80.498,A -85,B 0,C 180,E1 -11334.925,E2 -11334.925} C_VEL
LIN {X 0,Y 397.449,Z 80.465,A -85,B 0,C 180,E1 -11337.973,E2 -11337.973} C_VEL
LIN {X 0,Y 397.578,Z 80.436,A -85,B 0,C 180,E1 -11339.999,E2 -11339.999} C_VEL
LIN {X 0,Y 397.375,Z 80.478,A -85,B 0,C 180,E1 -11343.041,E2 -11343.041} C_VEL
LIN {X 0,Y 397.364,Z 80.482,A -85,B 0,C 180,E1 -11347.111,E2 -11347.111} C_VEL
LIN {X 0,Y 397.221,Z 80.483,A -85,B 0,C 180,E1 -11350.19,E2 -11350.19} C_VEL
LIN {X 0,Y 397.225,Z 80.502,A -85,B 0,C 180,E1 -11353.32,E2 -11353.32} C_VEL
LIN {X 0,Y 397.18,Z 80.501,A -85,B 0,C 180,E1 -11357.155,E2 -11357.155} C_VEL
LIN {X 0,Y 397.107,Z 80.507,A -85,B 0,C 180,E1 -11360.729,E2 -11360.729} C_VEL
LIN {X 0,Y 397.131,Z 80.513,A -85,B 0,C 180,E1 -11364.018,E2 -11364.018} C_VEL
LIN {X 0,Y 397.192,Z 80.492,A -85,B 0,C 180,E1 -11367.39,E2 -11367.39} C_VEL
LIN {X 0,Y 397.077,Z 80.526,A -85,B 0,C 180,E1 -11370.882,E2 -11370.882} C_VEL
LIN {X 0,Y 397.123,Z 80.504,A -85,B 0,C 180,E1 -11374.493,E2 -11374.493} C_VEL
LIN {X 0,Y 397.106,Z 80.521,A -85,B 0,C 180,E1 -11378.274,E2 -11378.274} C_VEL
LIN {X 0,Y 397.109,Z 80.51,A -85,B 0,C 180,E1 -11380.905,E2 -11380.905} C_VEL
LIN {X 0,Y 397.099,Z 80.519,A -85,B 0,C 180,E1 -11383.648,E2 -11383.648} C_VEL
LIN {X 0,Y 397.098,Z 80.494,A -85,B 0,C 180,E1 -11386.521,E2 -11386.521} C_VEL
LIN {X 0,Y 397.111,Z 80.511,A -85,B 0,C 180,E1 -11390.423,E2 -11390.423} C_VEL
LIN {X 0,Y 397.106,Z 80.502,A -85,B 0,C 180,E1 -11394.265,E2 -11394.265} C_VEL
LIN {X 0,Y 397.111,Z 80.509,A -85,B 0,C 180,E1 -11396.727,E2 -11396.727} C_VEL
LIN {X 0,Y 397.121,Z 80.502,A -85,B 0,C 180,E1 -11400.296,E2 -11400.296} C_VEL
LIN {X 0,Y 397.191,Z 80.51,A -85,B 0,C 180,E1 -11402.61,E2 -11402.61} C_VEL
LIN {X 0,Y 397.13,Z 80.52,A -85,B 0,C 180,E1 -11405.982,E2 -11405.982} C_VEL
LIN {X 0,Y 397.135,Z 80.519,A -85,B 0,C 180,E1 -11409.704,E2 -11409.704} C_VEL
LIN {X 0,Y 397.178,Z 80.512,A -85,B 0,C 180,E1 -11412.845,E2 -11412.845} C_VEL
LIN {X 0,Y 397.223,Z 80.507,A -85,B 0,C 180,E1 -11416.679,E2 -11416.679} C_VEL
LIN {X 0,Y 397.215,Z 80.509,A -85,B 0,C 180,E1 -11419.809,E2 -11419.809} C_VEL
LIN {X 0,Y 397.361,Z 80.491,A -85,B 0,C 180,E1 -11422.888,E2 -11422.888} C_VEL
LIN {X 0,Y 397.253,Z 80.504,A -85,B 0,C 180,E1 -11424.925,E2 -11424.925} C_VEL
LIN {X 0,Y 397.46,Z 80.769,A -85,B 0,C 180,E1 -11428.227,E2 -11428.227} C_VEL
LIN {X 0,Y 397.651,Z 80.873,A -85,B 0,C 180,E1 -11430,E2 -11430} C_VEL
LIN {X 0,Y 397.378,Z 80.566,A -85,B 0,C 180,E1 -11433.041,E2 -11433.041} C_VEL
LIN {X 0,Y 397.361,Z 80.491,A -85,B 0,C 180,E1 -11437.112,E2 -11437.112} C_VEL
LIN {X 0,Y 397.215,Z 80.509,A -85,B 0,C 180,E1 -11440.191,E2 -11440.191} C_VEL
LIN {X 0,Y 397.223,Z 80.507,A -85,B 0,C 180,E1 -11443.321,E2 -11443.321} C_VEL
LIN {X 0,Y 397.178,Z 80.512,A -85,B 0,C 180,E1 -11447.155,E2 -11447.155} C_VEL
LIN {X 0,Y 397.099,Z 80.523,A -85,B 0,C 180,E1 -11450.73,E2 -11450.73} C_VEL
LIN {X 0,Y 397.13,Z 80.52,A -85,B 0,C 180,E1 -11454.018,E2 -11454.018} C_VEL
LIN {X 0,Y 397.131,Z 80.519,A -85,B 0,C 180,E1 -11456.317,E2 -11456.317} C_VEL
LIN {X 0,Y 396.46,Z 80.602,A -85,B 0,C 180,E1 -11457.164,E2 -11457.164} C_VEL
LIN {X 0,Y 393.586,Z 80.947,A -85,B 0,C 180,E1 -11458.54,E2 -11458.54} C_VEL
LIN {X 0,Y 391.149,Z 81.249,A -85,B 0,C 180,E1 -11459.651,E2 -11459.651} C_VEL
LIN {X 0,Y 390.097,Z 81.386,A -85,B 0,C 180,E1 -11460.511,E2 -11460.511} C_VEL
LIN {X 0,Y 390.009,Z 81.395,A -85,B 0,C 180,E1 -11460.802,E2 -11460.802} C_VEL
LIN {X 0,Y 390.064,Z 81.371,A -85,B 0,C 180,E1 -11464.025,E2 -11464.025} C_VEL
LIN {X 0,Y 390.042,Z 81.4,A -85,B 0,C 180,E1 -11467.552,E2 -11467.552} C_VEL
LIN {X 0,Y 390.052,Z 81.373,A -85,B 0,C 180,E1 -11470.822,E2 -11470.822} C_VEL
LIN {X 0,Y 390.051,Z 81.378,A -85,B 0,C 180,E1 -11473.886,E2 -11473.886} C_VEL
LIN {X 0,Y 390.077,Z 81.392,A -85,B 0,C 180,E1 -11477.62,E2 -11477.62} C_VEL
LIN {X 0,Y 390.091,Z 81.388,A -85,B 0,C 180,E1 -11480.909,E2 -11480.909} C_VEL
LIN {X 0,Y 390.083,Z 81.385,A -85,B 0,C 180,E1 -11484.794,E2 -11484.794} C_VEL
LIN {X 0,Y 390.021,Z 81.401,A -85,B 0,C 180,E1 -11488.496,E2 -11488.496} C_VEL
LIN {X 0,Y 390.115,Z 81.376,A -85,B 0,C 180,E1 -11492.071,E2 -11492.071} C_VEL
LIN {X 0,Y 390.078,Z 81.393,A -85,B 0,C 180,E1 -11495.52,E2 -11495.52} C_VEL
LIN {X 0,Y 390.061,Z 81.388,A -85,B 0,C 180,E1 -11498.879,E2 -11498.879} C_VEL
LIN {X 0,Y 390.126,Z 81.371,A -85,B 0,C 180,E1 -11502.167,E2 -11502.167} C_VEL
LIN {X 0,Y 390.146,Z 81.384,A -85,B 0,C 180,E1 -11505.393,E2 -11505.393} C_VEL
LIN {X 0,Y 390.157,Z 81.369,A -85,B 0,C 180,E1 -11508.572,E2 -11508.572} C_VEL
LIN {X 0,Y 390.343,Z 81.346,A -85,B 0,C 180,E1 -11511.994,E2 -11511.994} C_VEL
LIN {X 0,Y 390.226,Z 81.375,A -85,B 0,C 180,E1 -11514.834,E2 -11514.834} C_VEL
LIN {X 0,Y 390.417,Z 81.34,A -85,B 0,C 180,E1 -11517.937,E2 -11517.937} C_VEL
LIN {X 0,Y 390.548,Z 81.311,A -85,B 0,C 180,E1 -11520.001,E2 -11520.001} C_VEL
LIN {X 0,Y 390.31,Z 81.36,A -85,B 0,C 180,E1 -11523.097,E2 -11523.097} C_VEL
LIN {X 0,Y 390.338,Z 81.358,A -85,B 0,C 180,E1 -11526.202,E2 -11526.202} C_VEL
LIN {X 0,Y 390.315,Z 81.346,A -85,B 0,C 180,E1 -11528.283,E2 -11528.283} C_VEL
LIN {X 0,Y 390.171,Z 81.375,A -85,B 0,C 180,E1 -11532.484,E2 -11532.484} C_VEL
LIN {X 0,Y 390.14,Z 81.382,A -85,B 0,C 180,E1 -11535.677,E2 -11535.677} C_VEL
LIN {X 0,Y 390.106,Z 81.366,A -85,B 0,C 180,E1 -11538.923,E2 -11538.923} C_VEL
LIN {X 0,Y 390.048,Z 81.394,A -85,B 0,C 180,E1 -11542.234,E2 -11542.234} C_VEL
LIN {X 0,Y 390.12,Z 81.375,A -85,B 0,C 180,E1 -11545.744,E2 -11545.744} C_VEL
LIN {X 0,Y 390.06,Z 81.392,A -85,B 0,C 180,E1 -11549.11,E2 -11549.11} C_VEL
LIN {X 0,Y 390.044,Z 81.394,A -85,B 0,C 180,E1 -11552.722,E2 -11552.722} C_VEL
LIN {X 0,Y 390.057,Z 81.392,A -85,B 0,C 180,E1 -11555.826,E2 -11555.826} C_VEL
LIN {X 0,Y 390.068,Z 81.388,A -85,B 0,C 180,E1 -11559.218,E2 -11559.218} C_VEL
LIN {X 0,Y 390.044,Z 81.4,A -85,B 0,C 180,E1 -11562.374,E2 -11562.374} C_VEL
LIN {X 0,Y 390.046,Z 81.395,A -85,B 0,C 180,E1 -11565.355,E2 -11565.355} C_VEL
LIN {X 0,Y 390.033,Z 81.393,A -85,B 0,C 180,E1 -11568.187,E2 -11568.187} C_VEL
LIN {X 0,Y 390.092,Z 81.38,A -85,B 0,C 180,E1 -11570.908,E2 -11570.908} C_VEL
LIN {X 0,Y 390.088,Z 81.381,A -85,B 0,C 180,E1 -11574.794,E2 -11574.794} C_VEL
LIN {X 0,Y 390.029,Z 81.395,A -85,B 0,C 180,E1 -11578.496,E2 -11578.496} C_VEL
LIN {X 0,Y 390.15,Z 81.624,A -85,B 0,C 180,E1 -11579.774,E2 -11579.774} C_VEL
